//Dozownik 12 (druga faza)                                       			                    
lrDispencer1DoseVolumeShow							:   ST_LrParametr;	 //:=300; 			    // Objętość do wydozowania [ml]
lrDispencer1Phase1VolumeShow						:   ST_LrParametr;	//:=100;			    // Objętość fazy początkowej [ml]
lrDispencer1Phase2VolumeShow						:   ST_LrParametr;	//:=200;			    // Objętość fazy końcowej [ml]
lrDispencer1Phase1VelocityShow						:   ST_LrParametr;	//:=500;			    // Prędkość fazy początkowej [ml/s]
lrDispencer1Phase2VelocityShow						:   ST_LrParametr;	//:=500;			    // Prędkość fazy dozowania [ml/s]
lrDispencer1Phase3VelocityShow						:   ST_LrParametr;	//:=500;			    // Prędkość fazy koncowej [ml/s]
lrDispencer1SuckVelocityShow						:   ST_LrParametr;	//:=500;			    // Prędkość zasysania masy [ml/s2]
lrDispencer1Phase1AccelerationShow					:   ST_LrParametr;	//:=3000;			    // Przyśpieszenie fazy początkowej [ml/s2]
lrDispencer1Phase2AccelerationShow					:   ST_LrParametr;	//:=3000;			    // Przyśpieszenie fazy dozowania [ml/s2]
lrDispencer1Phase3AccelerationShow					:   ST_LrParametr;	//:=3000;			    // Przyśpieszenie fazy końcowej [ml/s2]
lrDispencer1SuckAccelerationShow					:   ST_LrParametr;	//:=3000;			    // Przyśpieszenie zasysania masy [ml/s2]
lrDispencer1Phase1DecelerationShow					:   ST_LrParametr;	//:=3000;			    // Dynamika zwalniania w fazie początkowej
lrDispencer1Phase2DecelerationShow					:   ST_LrParametr;	//:=3000;			    // Dynamika zwalniania dozowania
lrDispencer1Phase3DecelerationShow					:   ST_LrParametr;	//:=3000;			    // Dynamika zwalniania fazy końcowej
udiDispencer1DosingDoneDelayTimeShow				:	ST_UdiParametr; //:=0; 				    // Zwłoka po wydozowaniu
lrDispencer1SuckValveOpenVolumeShow					:   ST_LrParametr;	//:=0;				    // Objętość przy której otwiera się zawór ssania [3] 
lrDispencer1SuckValveOpenTimeDelayShow				:   ST_LrParametr;	//:=0;				    // Zwłoka rozpoczęcia ssania po tłoczeniu [ms] [3]
lrDispencer1SuckValveCloseVolumeShow				:   ST_LrParametr;	//:=0;				    // [H] Objętość zamknięcia zaworu ssania od końca ssania [4]
lrDispencer1SuckValveCloseTimeDelayShow				:   ST_LrParametr;	//:=0;				    // Zwłoka zamknięcia zaworu ssącego [ms] [4] 
lrDispencer1DoseValveOpenVolumeShow					:   ST_LrParametr;	//:=0;				    // [H] Objętość przy której otwiera się zawór tłoczenia [ml] [1]
lrDispencer1DoseValveOpenTimeAccShow				:   ST_LrParametr;	//:=0;				    // Wyprzedzenie otwarcia zaworu tłoczenia [1] [ms]
lrDispencer1DoseValveCloseVolumeShow				:   ST_LrParametr;	//:=0;				    // Pozostała objętość dozy - zamknięcie zaworu tłoczenia [ml] [2]
lrDispencer1DoseValveCloseTimeDecShow				:   ST_LrParametr;	//:=0;				    // Zwłoka zamkniecia zaworu tłoczenia [2] [ms]
lrDispencer1DoseSuckingVolumeShow					:   ST_LrParametr;	//:=0;				    // Ilość dozy do posysenia [ml]	[5] [Podsysanie] 
lrDispencer1DoseSuckingTimeDelayShow				:   ST_LrParametr;	//:=0;				    // Opóźnienie podsysania [ms] [6] [Podsysanie] 
bDispencer1DoseSuckingShow							:	ST_BoolParametr;				        // Aktywacja podsysania
bDispencer1LiftSynchroPh1Show						:	ST_BoolParametr;				        // Synchronizacja z podnosnikiem w fazie początkowej
bDispencer1LiftSynchroPh2Show						:	ST_BoolParametr;				        // Synchronizacja z podnosnikiem w fazie dozowania
bDispencer1LiftSynchroPh3Show						:	ST_BoolParametr;				        // Synchronizacja z podnosnikiem w fazie końcowej
lrDispencer1LifterStartDosePositionShow				:   ST_LrParametr;	//:=20;				    // Pozycja rozpoczęcia dozowania
lrDispencer1LifterStopDosePositionShow				:   ST_LrParametr;	//:=60;				    // Pozycja zakończenia dozowania
lrDispencer1LifterVelocityShow						:   ST_LrParametr;	//:=100;			    // [H] Prędkość podnośnika 
lrDispencer1LifterAccelerationShow					:   ST_LrParametr;	//:=2;				    // [H] Przyspieszenie podnośnika
lrDispencer1LifterDecelerationShow					:   ST_LrParametr;	//:=2;				    // [H] Zwalnianie podnośnika
                                                                                                
//Dozowniki 34 (pierwsza faza)                                                                  		
lrDispencer2DoseVolumeShow							:   ST_LrParametr;	//:=300; 			    // Objętość do wydozowania                                           
lrDispencer2Phase1VolumeShow						:   ST_LrParametr;	//:=100;			    // Objętość fazy początkowej                                         
lrDispencer2Phase2VolumeShow						:   ST_LrParametr;	//:=200;			    // Objętość fazy końcowej                                            
lrDispencer2Phase1VelocityShow						:   ST_LrParametr;	//:=500;			    // Prędkość fazy początkowej                                         
lrDispencer2Phase2VelocityShow						:   ST_LrParametr;	//:=500;			    // Prędkość fazy dozowania                                           
lrDispencer2Phase3VelocityShow						:   ST_LrParametr;	//:=500;			    // Prędkość fazy koncowej                                            
lrDispencer2SuckVelocityShow						:   ST_LrParametr;	//:=500;			    // Prędkość zasysania masy                                           
lrDispencer2Phase1AccelerationShow					:   ST_LrParametr;	//:=3000;			    // Przyspieszenie fazy początkowej                                   
lrDispencer2Phase2AccelerationShow					:   ST_LrParametr;	//:=3000;			    // Przyspieszenie fazy dozowania                                     
lrDispencer2Phase3AccelerationShow					:   ST_LrParametr;	//:=3000;			    // Przyspieszenie fazy końcowej                                      
lrDispencer2SuckAccelerationShow					:   ST_LrParametr;	//:=3000;			    // Przyspieszenie zasysania masy                                     
lrDispencer2Phase1DecelerationShow					:   ST_LrParametr;	//:=3000;			    // Dynamika zwalniania w fazie początkowej                           
lrDispencer2Phase2DecelerationShow					:   ST_LrParametr;	//:=3000;			    // Dynamika zwalniania dozowania                                     
lrDispencer2Phase3DecelerationShow					:   ST_LrParametr;	//:=3000;			    // Dynamika zwalniania fazy końcowej                                 
udiDispencer2DosingDoneDelayTimeShow				:	ST_UdiParametr; //:=0; 				    // Zwłoka po wydozowaniu                                             
lrDispencer2SuckValveOpenVolumeShow					:   ST_LrParametr;	//:=0;				    // Objętość przy której otwiera się zawór ssania [3]                 
lrDispencer2SuckValveOpenTimeDelayShow				:   ST_LrParametr;	//:=0;				    // Zwłoka rozpoczęcia ssania po tłoczeniu [ms] [3]                   
lrDispencer2SuckValveCloseVolumeShow				:   ST_LrParametr;	//:=0;				    // [H] Objętość zamknięcia zaworu ssania od końca ssania [4]    
lrDispencer2SuckValveCloseTimeDelayShow				:   ST_LrParametr;	//:=0;				    // Zwłoka zamknięcia zaworu ssącego [ms] [4]                         
lrDispencer2DoseValveOpenVolumeShow					:   ST_LrParametr;	//:=0;				    // [H] Objętość przy której otwiera się zawór tłoczenia [ml] [1]
lrDispencer2DoseValveOpenTimeAccShow				:   ST_LrParametr;	//:=0;				    // Wyprzedzenie otwarcia zaworu tłoczenia [1] [ms]                   
lrDispencer2DoseValveCloseVolumeShow				:   ST_LrParametr;	//:=0;				    // Pozostała objętość dozy - zamknięcie zaworu tłoczenia [ml] [2]    
lrDispencer2DoseValveCloseTimeDecShow				:   ST_LrParametr;	//:=0;				    // Zwłoka zamkniecia zaworu tłoczenia [2] [ms]                       
lrDispencer2DoseSuckingVolumeShow					:   ST_LrParametr;	//:=0;				    // Ilość dozy do posysenia [ml]	[5] [Podsysanie]                     
lrDispencer2DoseSuckingTimeDelayShow				:   ST_LrParametr;	//:=0;				    // Opóźnienie podsysania [ms] [6] [Podsysanie]                       
bDispencer2DoseSuckingShow							:	ST_BoolParametr;				        // Aktywacja podsysania                                              
bDispencer2LiftSynchroPh1Show						:	ST_BoolParametr;				        // Synchronizacja z podnosnikiem w fazie początkowej                 
bDispencer2LiftSynchroPh2Show						:	ST_BoolParametr;				        // Synchronizacja z podnosnikiem w fazie dozowania                   
bDispencer2LiftSynchroPh3Show						:	ST_BoolParametr;			            // Synchronizacja z podnosnikiem w fazie końcowej                    
lrDispencer2LifterStartDosePositionShow				:   ST_LrParametr;	//:=20;				    // Pozycja rozpoczęcia dozowania                                     
lrDispencer2LifterStopDosePositionShow				:   ST_LrParametr;	//:=60;				    // Pozycja zakończenia dozowania                                     
lrDispencer2LifterVelocityShow						:   ST_LrParametr;	//:=100;			    // [H] Prędkość podnośnika                                      
lrDispencer2LifterAccelerationShow					:   ST_LrParametr;	//:=2;				    // [H] Przyspieszenie podnośnika                                
lrDispencer2LifterDecelerationShow					:   ST_LrParametr;	//:=2;				    // [H] Zwalnianie podnośnika                                    
                                                        		                                
//Chwytak dozowników 1234                                                                       
bDispencersCatchEnableShow	      					:	ST_BoolParametr;			            // [H] Aktywacja    
bDispencersCatchMaxPressureShow	      				:	ST_BoolParametr;			            // Zwiększona siła chwytania            		
lrDispencersCatchHeightSVShow						:   ST_LrParametr;	//:=86;  			    // Pozycja chwytaka
//Kalibracja chwytaków 1234                                                                     
lrDispencersCatch1ClosedValueShow                   :   ST_LrParametr;	                        // Chwytak 1 | wartość kalibracji zamkniętego chwytaka
lrDispencersCatch1OpenValueShow                     :   ST_LrParametr;	                        // Chwytak 1 | wartość kalibracji otwartego chwytaka
lrDispencersCatch2ClosedValueShow                   :   ST_LrParametr;	                        // Chwytak 2 | wartość kalibracji zamkniętego chwytaka
lrDispencersCatch2OpenValueShow                     :   ST_LrParametr;	                        // Chwytak 2 | wartość kalibracji otwartego chwytaka
lrDispencersCatch3ClosedValueShow                	:   ST_LrParametr;	                        // Chwytak 3 | wartość kalibracji zamkniętego chwytaka
lrDispencersCatch3OpenValueShow                     :   ST_LrParametr;	                        // Chwytak 3 | wartość kalibracji otwartego chwytaka
lrDispencersCatch4ClosedValueShow                   :   ST_LrParametr;	                        // Chwytak 4 | wartość kalibracji zamkniętego chwytaka
lrDispencersCatch4OpenValueShow                     :   ST_LrParametr;	                        // Chwytak 4 | wartość kalibracji otwartego chwytaka
lrDispencersCatchToleranceShow                      :   ST_LrParametr;	                        // Tolerancja chwytaka [0-100%]      
                                          		                                                
//Zbiorniki                                                                                     
bTank1MixerEnableShow								:	ST_BoolParametr;	   				    // Mieszadło
bTankHeatingEnableShow								:	ST_BoolParametr;				        // Grzanie                                     		
iTankHeatingTempSVShow								:	ST_DIParametrr;							// Temperatura
bTank1PressureEnableShow							:	ST_BoolParametr;				        // Ciśnienie                                   		
bTank1SupplyPumpEnableShow							:	ST_BoolParametr;			            // Aktywacja pompy 1
bTank2SupplyPumpEnableShow							:	ST_BoolParametr;			            // Aktywacja pompy 2
uTank1LevelSetpointShow								:	ST_UdiParametr;						    // [H] Wartość zadana masy do czujnika poziomu w zbiorniku nr 1
uTank2LevelSetpointShow								:	ST_UdiParametr;						    // [H] Wartość zadana masy do czujnika poziomu w zbiorniku nr 2
bTank1LevelSignalInvertShow							:	ST_BoolParametr;			            // [H] Odwróć sygnał z czujnika zbiornika pierwszego
bTank2LevelSignalInvertShow							:	ST_BoolParametr;			            // [H] Odwróć sygnał z czujnika zbionirka drugiego
                                        			                                            
//Waga                                           			                                    
bWeight1EnableShow									:	ST_BoolParametr;	                    // Aktywacja
lrWeightMassSVShow 									:   ST_LrParametr;						    // Waga zadana 
iWeight1ActuatorUpDelayShow							:	ST_DIParametrr;						    // Opóźnienie podnoszenia wagi 1
iWeight2ActuatorUpDelayShow							:	ST_DIParametrr;						    // Opóźnienie podnoszenia wagi 2
iWeight3ActuatorUpDelayShow							:	ST_DIParametrr;					        // Opóźnienie podnoszenia wagi 3
iWeight4ActuatorUpDelayShow							:	ST_DIParametrr;							// Opóźnienie podnoszenia wagi 4
iWeight5ActuatorUpDelayShow							:	ST_DIParametrr;						    // Opóźnienie podnoszenia wagi 5 
iWeight6ActuatorUpDelayShow							:	ST_DIParametrr;				            // Opóźnienie podnoszenia wagi 6
                                                                                                
//Korekcja wagi                                     			                                
lrFormWeightShow 									:   ST_LrParametr;						    // [H] Waga formatki
lrMass1DensityShow									:   ST_LrParametr;					        // [H] Gęstoć masy pierwszej fazy [g/ml]
lrMass2DensityShow									:   ST_LrParametr;					        // [H] Gęstoć masy drugiej fazy [g/ml]
lrCupWeightShow										:   ST_LrParametr;						    // Waga opakowania (z platynką, zależnie od opakowania) [g]
lrWholePackageWeightShow							:   ST_LrParametr;						    // [H] Waga całego opakowania bez masy (kubeczek,platynka,nakrętka) [g]
lrWeight1MeasurmentCorrectionShow					:   ST_LrParametr;					        // [H] Korekta wagi zmierzonej [g] , różnica pomiedzy wskazaniami wagi zewnętrznej a linią
bDispencer1WeightCorrectionEnableShow				:	ST_BoolParametr;			            // Aktywacja korekcji 1
bDispencer2WeightCorrectionEnableShow				:	ST_BoolParametr;				        // Aktywacja korekcji 2
bDispencer3WeightCorrectionEnableShow				:	ST_BoolParametr;			            // Aktywacja korekcji 3
bDispencer4WeightCorrectionEnableShow				:	ST_BoolParametr;			            // Aktywacja korekcji 4	
lrWeightUpperToleranceShow							:   ST_LrParametr;				            // Górny zakres wagi [g]
lrWeightLowerToleranceShow							:   ST_LrParametr;					        // Dolny zakres wagi [g]
iWeightCorrectionNumberOfSamplesShow				:	ST_UdiParametr;		//:=2;				// Ilość próbek korekcji [x] (1-20)
                                                                                                
//Podajnik platynek                                                                             
bLidFeederEnableShow								:	ST_BoolParametr;			            // Zezwolenie na pracę podajnika platynek 
bLidFeederHeaterEnableShow							:	ST_BoolParametr;		                // Zezwolenie na prace grzałki podajnika platynek 
lrLidFeederHeightPosSVShow							:   ST_LrParametr;						    // Wysokość na której ma znajdować się podajnik platynek
iLidFeederHeatingTimeShow							:	ST_DIParametrr;						    // Czas zgrzewania wstępnego podajnika platynek [ms]
iLidFeederTempHisteresisShow						:	ST_DIParametrr;					        // Histereza poprawnej temperatury grzałki podajnika platynek 1 (+/- *C), po jej przekrocz
iLidFeeder1TempSVShow								:	ST_DIParametrr;						    // Temperatura zadana grzałki podajnika platynek 1
iLidFeeder2TempSVShow								:	ST_DIParametrr;					        // Temperatura zadana grzałki podajnika platynek 2
                                                                                                
//Przeciąganie podajnika platynek                                                               
bLidFeederDragingStationEnableShow					:	ST_BoolParametr;			            // Aktywacja przeciagania formatek pod podajnikem płatynek
lrLidFeederDragingStationVelocityShow				:   ST_LrParametr;	 				        // Prędkosć przeciągania formatek pod podajnikem płatynek [0-100 %]	
lrLidFeederDragingStationAccelerationShow			:   ST_LrParametr;	 				        // Przyspieszenie przeciągania formatek pod podajnikem płatynek 	
lrLidFeederDragingStationDecelerationShow			:   ST_LrParametr;	 				        // Zmniejszenie prędkości przeciągania formatek pod podajnikem płatynek 	
                                                                                                
//Sprawdzanie platynek                                                                          
bLidPuttedCheckEnableShow      						:	ST_BoolParametr;			            	// Zezwolenie na prace stacji sprawdzania nakrętek
lrLidPuttedCheckHeightSVShow 	 					:   ST_LrParametr;	            	        	
lrLidPuttedCheckPositionShow						:   ST_LrParametr;					        	// Pozycka sprawdzania platynki
lrLidPuttedCheckAreaShow							:   ST_LrParametr;					        	// [-50...50]  lrLidPuttedCheckPosition +- lrLidPuttedCheckArea. Granica monitorowania
iLidPuttedCheckProgramShow							:	ST_DIParametrr;								// Program czujnika wizyjnego 0-20
                                                                                                
//Zgrzewanie                                                                                    
bLidSealerEnableShow								:	ST_BoolParametr;			            // Zezwolenie na pracę podajnika 
bLidSealerHeaterEnableShow							:	ST_BoolParametr;			            // Zezwolenie na prace grzałki  
iLidSealerHeatingTimeShow							:	ST_DIParametrr;						    // Czas zgrzewania  [ms]
lrLidSealerPressureShow								:   ST_LrParametr;					        //	Siła zgrzewania [kg] 
lrLidSealerHeightPosSVShow							:   ST_LrParametr;					        // Wysokoć na której ma znajdować się grzałka
iLidSealerTempHisteresisShow						:	ST_DIParametrr;							// Histereza poprawnej temperatury grzałki (+/- *C), po jej przekroczeniu grzałka wpada w 
iLidSealer1TempSVShow								:	ST_DIParametrr;					        // Temperatura zadana grzałki 1                                                           
iLidSealer2TempSVShow								:	ST_DIParametrr;				            // Temperatura zadana grzałki 2
                                                                                                
//Przeciąganie zgrzewania                                                                       
bLidSealerDragingStationEnableShow					:	ST_BoolParametr;			            // Aktywacja przeciagania formatek pod zakrecarkami
lrLidSealerDragingStationVelocityShow				:   ST_LrParametr;				            // Prędkosć przeciągania formatek pod zakręcarkami [0-100 %]
lrLidSealerDragingStationAccelerationShow			:   ST_LrParametr;	 				        // Przyspieszenie przeciągania formatek pod podajnikem płatynek 	
lrLidSealerDragingStationDecelerationShow			:   ST_LrParametr;					        // Zmniejszenie prędkości przeciągania formatek pod podajnikem płatynek 	
                                                                                                
//Szlaban podawania zamknięć                            				                        
bCapFeederGateEnableShow							:	ST_BoolParametr;		                // Aktywacja 
iCapFeederGateBlockingTimeShow						:	ST_DIParametrr;							// Czas blokowania
                                                                                                
//[H] Podajnik zamknięć                        				                                    
bCapFeederEnableShow								:	ST_BoolParametr;		                // [H] Aktywacja
lrCapFeederHeightPosSVShow							:   ST_LrParametr;	//:=140;			    // [H] Pozycja
iCapFeederTimeDelayOnShow							:	ST_DIParametrr;						    // [H] Opóźnienie włączenia
iCapFeederTimeDelayOffShow							:	ST_DIParametrr;						    // [H] Opóźnienie wyłączenia
iCapFeederTimeToEmptySleeveErrorShow				:	ST_DIParametrr;						    // [H] Czas do alarmu pustego rękawa [s] (10-120 s)
                                                                                                
//Sorter nasadek                                                                                
//Zmienne z innego sterownika                                                                   
bCapSorterOnlyWeightOKEnableShow					:	ST_BoolParametr;		                // Nakładanie zamknięć tylko na opakowania z waga OK
                                                                                                
//Przeciąganie pod sorterem nasadek                                                             
bCapSorterDragEnableShow							:	ST_BoolParametr;		                // [H] Aktywacja
lrCapSorterDragVelocityShow							:   ST_LrParametr;					        // Prędkość
lrCapSorterDragAccelerationShow						:   ST_LrParametr;						    // Przyspieszenie 
lrCapSorterDragDecelerationShow						:   ST_LrParametr;					        // Hamowanie
                             				                                                    
//Sprawdzanie nasadki                                      				                        
bCapPuttedCheckEnableShow							:	ST_BoolParametr;			            // Aktywacja
lrCapPuttedCheckHeightPosSVShow						:   ST_LrParametr;	//:=69;				    // Pozycja
                             					                                                
//Zakrecarka szczekowa (Zachować kolejność i opisy!)                                            
bGripperScrewer1EnableShow							:	ST_BoolParametr;			            // Aktywacja 1
lrGripperScrewingTightTorqueShow					:   ST_LrParametr;	  				        // Nastawa momentu zakręcania [Nm]
bGripperScrewer2EnableShow							:	ST_BoolParametr;		                // Aktywacja 2
lrGripperScrewing2TightTorqueShow					:   ST_LrParametr;	  				        // Nastawa momentu zakręcania 2 [Nm]
iGripperScrewer1ToolShow							:	ST_DIParametrr;					        // Wybór narzędzia (1-5), opisy w tablicy AsGripperScrewerTool	
lrGripperScrewer1VelocityShow						:   ST_LrParametr;	//:=6000; 			    // Prędkość zakręcania [rpm]
nGripperScrewer1TightTimeShow						:	ST_DiParametrr; //:=100;  			    // Czas przytrzymania podczas dokręcania [ms] 	
iGripperScrewer1StartDelayShow						:	ST_DIParametrr;					        // Zwoka przed zakręcaniem			
lrGripperScrewerReadyPositionShow					:   ST_LrParametr;	 //:= 250;  		    // Pozycja gotowości
lrGripperScrewerPushingCapPositionShow				:   ST_LrParametr;	//:= 250;  		        // Pozycja docisku  
lrGripperScrewerScrewingCapPositionShow				:   ST_LrParametr;	//:= 250;  		        // Pozycja zakręcania	
lrGripperScrewerPressureShow						:   ST_LrParametr;						    // Siła chwytaka nasadki (0.0 kg)
lrGripperScrewerCatchPressureShow 					:   ST_LrParametr;						    // Siła chwytaka butelki (0.0 kg)
lrDispencerCatchPressureShow 						:   ST_LrParametr;						    // Siła chwytaka butelki pod dozownikami (0.0 kg)
lrGripperScrewerPressureExhaustLevelShow			:   ST_LrParametr;						    // Prędkość zamykania chwytaka nasadki (0.0-100.0 %)
lrGripperScrewerCatchPressureExhaustLevelShow		:   ST_LrParametr;						    // Prędkość zamykania chwytaka opakowania (0.0-100.0 %)
lrGripperScrewerTurnoversToFullScrewedShow			:   ST_LrParametr;						    // Opakowanie | Ilość obrotów zamknięcia [obr.] (0.5-10.0 obr.)
lrGripperScrewerThreadPitchShow						:   ST_LrParametr;						    // Opakowanie | Skok gwintu [mm] (0.1-10.0 mm)
lrGripperScrewerThreadTimesShow						:   ST_LrParametr;						    // Opakowanie | Krotność gwintu [x] (1-10 x)                       		
nGripperScrewerCatchHeightSVShow					:	ST_DiParametrr; //:=86;  				// Pozycja chwytaka opakowań
bGripperScrewer1FindScrewShow						:	ST_BoolParametr;			            // Szukanie gwintu w pozycji zakręcania	
bGripperScrewer1Option4Show							:	ST_BoolParametr;			            // Szukanie gwintu w pozycji dociskania	
lrGripperScrewer1FindingScrewDegreeShow				:   ST_LrParametr;	 				        // Kąt szukania gwintu (max. dla opcji szukania gwintu z czuj. wys.)	
bGripperScrewer1Option1Show							:	ST_BoolParametr;		                // Otwarty chwytak przy szukaniu gwintu	
bGripperScrewer1Option2Show							:	ST_BoolParametr;			            // Obrót do tyłu w pozycji dociskania (w trakcie przejazdu do poz. doc.)
bGripperScrewer1Option3Show							:	ST_BoolParametr;			            // Dodatkowy ruch chwytakiem przed zakręceniem  (w poz. doc.)	
bGripperScrewer1Option5Show							:	ST_BoolParametr;			            // Szukanie gwintu z czujnikiem wysokości
bGripperScrewer1Option6Show							:	ST_BoolParametr;			            // Obrót z pozycji docisku do zakręcania
bGripperScrewer1Option7Show							:	ST_BoolParametr;		                // Tryb momentowy	
                                                                                                
//Przeciaganie formatek pod zakrecarkami                                                        
bBottleDragingStationEnableShow						:	ST_BoolParametr;			            // [H] Aktywacja 
lrBottleDragingStationVelocityShow					:   ST_LrParametr;					        // Prędkość
                                                                                                
//Sprawdzanie zakręcania                                                                        
bCapCorrectCheckEnableShow							:	ST_BoolParametr;				        // Aktywacja
lrCapCorrectCheckHeightPosSVShow					:   ST_LrParametr;	//:=69;				    // Pozycja
bCapCorrectCheckCameraEnableShow      				:	ST_BoolParametr;			            // Aktywacja sprawdzania orientacji nasadki
iCapCorrectCheckCameraProgramShow					:	ST_DIParametrr;			                // Program czujnika wizyjnego 0-20
                                                                                                
                                                                                                
//Robot butelek                                                                                 
bBottleTransferEnableShow							:	ST_BoolParametr;			            // Aktywacja
nBottleTransferProgramShow							:	ST_UdiParametr;						    // [H] Program robota	
iBottleTransferPickOffsetXShow 						:	ST_DIParametrr;					        // Offset X pozycji pobrania
iBottleTransferPickOffsetYShow 						:	ST_DIParametrr;							// Offset Y pozycji pobrania  
iBottleTransferPickOffsetZShow 						:	ST_DIParametrr;							// Offset Z pozycji pobrania
iBottleTransferPick2OffsetXShow						:	ST_DIParametrr;							// Offset X 2 pozycji pobrania	
iBottleTransferPick2OffsetYShow						:	ST_DIParametrr;					        // Offset Y 2 pozycji pobrania
iBottleTransferPick2OffsetZShow						:	ST_DIParametrr;							// Offset Z 2 pozycji pobrania
iBottleTransferPlace1OffsetXShow 					:	ST_DIParametrr;							// Offset X pozycji etykieciarki
iBottleTransferPlace1OffsetYShow 					:	ST_DIParametrr;							// Offset Y pozycji etykieciarki
iBottleTransferPlace1OffsetZShow 					:	ST_DIParametrr;						    // Offset Z pozycji etykieciarki
iBottleTransferPlace2OffsetXShow 					:	ST_DIParametrr;							// Offset X pozycji odrzutu
iBottleTransferPlace2OffsetYShow					:	ST_DIParametrr;							// Offset Y pozycji odrzutu	
iBottleTransferPlace2OffsetZShow 					:	ST_DIParametrr;							// Offset Z pozycji odrzutu
iBottleTransferSpeedShow							:	ST_DIParametrr;	  //:= 10;			    // Prędkość robota 	
bBottleTransferInkJetEnableShow						:	ST_BoolParametr;			            // Przesuwanie opakowania nad drukarką (Inkjet)
bBottleTransferPickOnlyOneShow						:	ST_BoolParametr;			            // [H] Pobieranie tylko 1 opakowania
bBottleTransferWeightEnableShow						:	ST_BoolParametr;				        // Przesuwanie opakowania na wagę 
iBottleTransferWeightIntervalShow					:	ST_DIParametrr;							// Interwał przesuwania na wagę
bBottleTransferRotateEnableShow						:	ST_BoolParametr;                        // Obrót orientacji nasadki   
                                                                                                
//Transporter odrzutu                      	                                                    
bBadBottleConveyorEnableShow						:	ST_BoolParametr;				        // [H] Aktywacja
nBadBottleConveyorVelocitySVShow					:	ST_UdiParametr;						    // Prędkość
                                                                                                
//Etykieciarka                                                                                  
bLabelMachineEnableShow								:	ST_BoolParametr;				        // Aktywacja
                                                                                                
//Stół odbierający                                                                              
bExitTurnTable1EnableShow							:	ST_BoolParametr;				        // Aktywacja
//Transporter odbierający                                                                       
bExitConveyorEnableShow								:	ST_BoolParametr;			            // Aktywacja
nExitConveyorVelocitySVShow							:	ST_UdiParametr;						    // Prędkość
                                                                                                
                                                                                                
//Transportery główne                                                                           
bFormTransportersEnableShow							:	ST_BoolParametr;				        // [H] Aktywacja
nFormTransportersDispencerVelocitySVShow			:	ST_UdiParametr;				            // Prędkość transportera przed dozownikami
nFormTransportersScrewerVelocitySVShow				:	ST_UdiParametr;				            // Prędkość transportera za dozownikami
nFormTransportersBeforeScrewerVelocitySVShow		:	ST_UdiParametr;			                // Prędkość transportera przed zakręcarką
nFormTransportersSlowerVelocitySVShow				:	ST_UdiParametr;				            // Prędkość spowalniacza 
                                                                                                
                                                                                                
//[H] InkJet obwodowy                                                                           
bCircularInkjetEnableShow							:	ST_BoolParametr;				        // [H] Aktywacja
iCircularInkjetSpeedShow							:	ST_DIParametrr;							// [H] Prędkość 
iCircularInkjetDelayShow							:	ST_DIParametrr;							// [H] Opóźnienie docisku rolek
iCircularInkjetHoldShow								:	ST_DIParametrr;							// [H] Czas przytrzymania [ms]

bROPPCappingEnableShow 								:	ST_BoolParametr;	
bROPPDragEnableShow 								:	ST_BoolParametr;	
bROPPFeederEnableShow 								:	ST_BoolParametr;	
bROPPSlowerEnableShow 								:	ST_BoolParametr;	
iROPPCapping1ToolShow 								:	ST_DIParametrr;	
iROPPCappingTime2Show 								:	ST_DIParametrr;	
iROPPCappingTimeShow 								:	ST_DIParametrr;	
iROPPFeederTimeDelayOffShow							:	ST_DIParametrr;	
iROPPFeederTimeDelayOnShow 							:	ST_DIParametrr;	
iROPPFeederTimeToEmptySleeveErrorShow 				:	ST_DIParametrr;	
lrROPPCappingHeightPosSVShow						:	ST_LrParametr;	
lrROPPCappingVelocitySVShow 						:	ST_LrParametr;	
lrROPPDragAccelerationShow 							:	ST_LrParametr;	
lrROPPDragDecelerationShow 							:	ST_LrParametr;	
lrROPPDragVelocityShow 								:	ST_LrParametr;	
lrROPPFeederHeightPosSVShow 						:	ST_LrParametr;	                                                                             
nROPPSlowerVelocitySVShow 							:	ST_UdiParametr;	

END_STRUCT                                                                                      
END_TYPE

// ---- POUs/Recipes/NewRecipes/ST_Recipe_UCF_PARAM.TcDUT
TYPE ST_Recipe_UCF_PARAM :
STRUCT
		//Sorter nasadek, typ produktu	
	iCapSorterProductType										:	ST_DIParametrr;		//:= 2; 		//		Typ produktu: 0- kule/fliptopy, 1- pompki, 2- disctop, 3-airless, 4-decoration cap (wyłączone podcisnienie na załapywarce), 5- decoration cap with new gripper (wyłączone podcisnienie + nowy program do robota)
	uiCapSorterIndexShow										:	ST_UdiParametr;	//:= 5;		//		Index produktu	
	bPresenceBottleEnableShow									:	ST_BoolParametr;					//		Sprawdzanie butelki w formatce

//--------------------------------------CapSorterTransporter-----------------------------------------------------------------------------------------------------------------------------	
	// Sorter nasadek, transporter zasobnika
	bCapSorterTransporterEnableShow								:	ST_BoolParametr;				//		Aktywacja
	iCapSorterTransporterTankConveyorVelocityShow				:	ST_DIParametrr;		//:= 1200;	//		Prędkość 							| [%] (1.0-100.0)
	iCapSorterTransporterStartDelayTimeShow						:	ST_DIParametrr;		//:= 100;		//		Timer do załączania 				| [ms] (0.0-10_000.0)
	udiCapSorterTransporterTimeProductOnSensorBeforeBrushShow	:	ST_UdiParametr;		//:= 150;		//		Timer pracy							| [ms] (0.0-10_000.0)
	iCapSorterTransporterEmptyingConveyorSpeedShow				:	ST_DIParametrr;		//:= 25;		// 		Prędkość, opróżnianie 				| [%] (1.0-100.0)
	iCapSorterTransporterVolumeOfCapsShow						:	ST_DIParametrr;		//:= 330;		//		Odłegłość do zamknięć, ostrzeżenie 	| [mm] (0.0-10_000.0)

//---------------------------------------CapSorterWheel----------------------------------------------------------------------------------------------------------------------------	
	// Sorter nasadek, stól
	bCapSorterWheelEnableShow									:	ST_BoolParametr;				//		Aktywacja
	lrCapSorterWheelMoveAccelerationEmptyTableShow				:   ST_LrParametr;			//:= 5000;	//		Dynamika rozpędzania - pusty 		| [obr/min²], (1.0-100_000.0) 
	lrCapSorterWheelMoveDecelerationEmptyTableShow				:   ST_LrParametr;			//:= 5000;    //		Dynamika spowalniania - pusty 		| [obr/min²] (1.0-100_000.0) 
	lrCapSorterWheelMoveSpeedEmptyTableShow						:   ST_LrParametr;		//:= 334;     //		Prędkość - pusty 					| [obr/min] (1.0-10_000.0)                
	lrCapSorterWheelMoveAngleEmptyTableShow						:   ST_LrParametr;			//:= 20;      //		Kąt - pusty 						| [obr/min] (0.0-360.0)                        
	lrCapSorterWheelJerkAngleEmptyTableShow						:   ST_LrParametr;		//:= 15000;   //		Zryw - pusty 						| [obr/min³] (1.0-1_000_000)                  
	iCapSorterWheelWaitingAfterRotationEmptyTableShow			:	ST_DIParametrr;		//:= 100;     //		Czas stabilizacji - pusty 			| [ms] (0.0-1_000)                 
	                                                                        //
	lrCapSorterWheelMoveAccelerationFullTableShow				:   ST_LrParametr;		//:= 5000;	//		Dynamika rozpędzania - pełny 		| [obr/min²], (1.0-100_000.0) 
	lrCapSorterWheelMoveDecelerationFullTableShow				:   ST_LrParametr;		//:= 5000;    //		Dynamika spowalniania - pełny 		| [obr/min²] (1.0-100_000.0) 
	lrCapSorterWheelMoveSpeedFullTableShow						:   ST_LrParametr;		//:= 334;     //		Prędkość - pełny 					| [obr/min] (1.0-10_000.0)                
	lrCapSorterWheelMoveAngleFullyTableShow						:   ST_LrParametr;			//:= 6;       //		Kąt - pełny 						| [obr/min] (0.0-360.0)                        
	lrCapSorterWheelJerkAngleFullTableShow						:   ST_LrParametr;			//:= 15000;   //		Zryw - pełny 						| [obr/min³] (1.0-1_000_000)                  
	iCapSorterWheelWaitingAfterRotationFullTableShow			:	ST_DIParametrr;		//:= 30;      //		Czas stabilizacji - pełny 			| [ms] (0.0-1_000)                 
	                                                                        //
	lrCapSorterWheelMoveAccelerationHalfFullTableShow			:   ST_LrParametr;			//:= 5000;	//		Dynamika rozpędzania - półpełny 	| [obr/min²], (1.0-100_000.0) 
	lrCapSorterWheelMoveDecelerationHalfFullTableShow			:   ST_LrParametr;			//:= 5000;    //		Dynamika spowalniania - półpełny 	| [obr/min²] (1.0-100_000.0) 
	lrCapSorterWheelMoveSpeedHalfFullTableShow					:   ST_LrParametr;			//:= 334;     //		Prędkość - półpełny 				| [obr/min] (1.0-10_000.0)                
	lrCapSorterWheelMoveAngleHalfFullyTableShow					:   ST_LrParametr;			//:= 12;      //		Kąt - półpełny						| [obr/min] (0.0-360.0)                        
	lrCapSorterWheelJerkAngleHalfFullTableShow					:   ST_LrParametr;			//:= 15000;   //		Zryw - półpełny 					| [obr/min³] (1.0-1_000_000)                  
	iCapSorterWheelWaitingAfterRotationHalfFullTableShow		:	ST_DIParametrr;		//:= 50;      //		Czas stabilizacji - półpełny 		| [ms] (0.0-1_000)                 

//-------------------------------------CapSorterCamera------------------------------------------------------------------------------------------------------------------------------	                                                    	
	// Sorter nasadek, system wizyjny
	
    bCapSorterCameraEnableShow									:	ST_BoolParametr;				//	[H]	Aktywacja                            	
	
//-----------------------------------------CapSorterRobot--------------------------------------------------------------------------------------------------------------------------	
	// Sorter nasadek, robot
	bCapSorterRobotEnableShow									:	ST_BoolParametr;				//		Aktywacja
                                                                                                                           	
	lrCapSorterRobotPlace1PositionXShow							:   ST_LrParametr;					//		Offset odkładania 1, X 			| [mm]	((-100.0)-100.0)       
	lrCapSorterRobotPlace1PositionYShow							:   ST_LrParametr;	    			//		Offset odkładania 1, Y 			| [mm]	((-100.0)-100.0)       
	lrCapSorterRobotPlace1PositionZShow							:   ST_LrParametr;	    			//		Offset odkładania 1, Z 			| [mm]	((-100.0)-100.0)       
	lrCapSorterRobotPlace1PositionCShow							:   ST_LrParametr;	    			//		Offset odkładania 1, C 			| [° ]	((-360.0)-360.0)                 
	iCapSorterRobotPickElevationShow							:	ST_DIParametrr;				//		Punkt nad poz. Pick				| [mm]	(30-1000)
	iCapSorterRobotPickTimeShow									:	ST_DIParametrr;					//		Czas przyssania					| [ms]	(0-10_000)
	iCapSorterRobotVacuumActivationShow							:	ST_DIParametrr;					//		Czas przed przyssaniem			| [ms]	(0-1000)
	iCapSorterRobotVacuumOffShow								:	ST_DIParametrr;					//		Czas przed oddmuchem			| [ms]	(0-1000)
	iCapSorterRobotPlaceTimeShow								:	ST_DIParametrr;					//		Czas oddmuchu					| [ms]	(0-1000)
	iCapSorterRobotTCP_PlaceOffsetShow							:	ST_DIParametrr;					//		Wysokość od TCP do p. odłożenia	| [mm]	(0-1000)									
	iCapSorterRobotAccelerationDecelerationShow					:	ST_DIParametrr;					//		Dynamika rozpędzania/hamowania	| [%]	(20-100)
	iCapSorterRobotGripperWatchdogShow							:	ST_DIParametrr;					//		Czas sprawdzania silownika		| [ms]	(0-1000)
	iCapSorterRobotParalaxCorrectionShow						:	ST_DIParametrr;				//		Korekta paralaxy				| [mm]	(0-100)
	
	iCapSorterRobotNumberToolShow								:	ST_DIParametrr;				//		Numer narzędzia					| 		(0-10)
	iCapSorterRobotPickPositionZShow							:	ST_DIParametrr;					//		Wysokość pobierania 			| [mm]	(0-200)
	iCapSorterRobotTCP_Lenght									:	ST_DIParametrr;					//		Długość chwytaka				| [mm]	(10-100)
	iCapSorterRobotProductDiametr								:	ST_DIParametrr;					//		Średnica nasadki				| [mm] 	(10-100)
	
//----------------------------------------CapSorterIntermediateTransporter---------------------------------------------------------------------------------------------------------------------------
	// Sorter nasadek, transporter zasypowy
	bCapSorterIntermediateTransporterEnableShow					:	ST_BoolParametr;			//		Aktywacja
	iCapSorterIntermediateTransporterAutoSpeedShow				:	ST_DIParametrr;		//:= 20;		//		Prędkość 					| [%] (1.0-100.0)
	iCapSorterIntermediateTransporterManualSpeedShow			:	ST_DIParametrr;		//:= 30;		//		Prędkość, manual 			| [%] (1.0-100.0)
	iCapSorterIntermediateTransporterEmptyingSpeedShow			:	ST_DIParametrr;		//:= 50;		//		Prędkość, opróżnianie 		| [%] (1.0-100.0)
	iCapSorterIntermediateTransporterDelayCountTimeShow			:	ST_DIParametrr;		//:= 100;		//		Timer pracy					| [ms]	(0.0-100_000.0)
	iCapSorterIntermediateTransporterReverseTimeShow			:	ST_DIParametrr;		//:= 4000;	//		Timer odwróconej pracy 		| [ms] (0.0-10_000.0)
	udiCapSorterIntermediateTransporterTimeProductOnSensorShow	:	ST_UdiParametr;		//:= 1800;	//		Czas produktu na czujniku 	| [ms] (0.0-10_000.0)	
	lrCapSorterIntermediateTransporterWheelAngleShow			:   ST_LrParametr;			//:= 6;		//		Kąt zasypu 					| [°] (1.0-360.0)
	
//----------------------------------------CapSorterIntermediateBrush---------------------------------------------------------------------------------------------------------------------------
	//Sorter nasadek, szczotka transportera
	bCapSorterIntermediateBrushEnableShow						:	ST_BoolParametr;				//		Aktywacja
	iCapSorterIntermediateBrushAutoSpeedShow					:	ST_DIParametrr;		//:= 30;		//		Prędkość  					| [%] (0.0-100.0)
	iCapSorterIntermediateBrushManualSpeedShow					:	ST_DIParametrr;		//:= 30;		//		Prędkość, manual 			| [%] (0.0-100.0)
	iCapSorterIntermediateBrushEmptyingSpeedShow				:	ST_DIParametrr;		//:= 30;		//		Prędkość, opróżnianie 		| [%] (0.0-100.0)
	lrCapSorterIntermediateBrushPositionHeightSVShow			:   ST_LrParametr;			//:= 45;		//		Wysokość 					| [mm] (0.0-10_000.0)

//----------------------------------------CapSorterBrush1OnWheel---------------------------------------------------------------------------------------------------------------------------
	// Sorter nasadek, szczotka stolu 1
	bCapSorterBrush1OnWheelEnableShow							:	ST_BoolParametr;					//		Aktywacja
	iCapSorterBrush1OnWheelAutoSpeedShow						:	ST_DIParametrr;		//:= 30;		//		Prędkość 					| [%] (0.0-100.0)
	iCapSorterBrush1OnWheelManualSpeedShow						:	ST_DIParametrr;		//:= 30;		//		Prędkość, manual 			| [%] (0.0-100.0)
	iCapSorterBrush1OnWheelEmptyingSpeedShow					:	ST_DIParametrr;		//:= 30;		//		Prędkość, opróżnianie 		| [%] (0.0-100.0)
	lrCapSorterBrush1OnWheelPositionHeightSVShow				:   ST_LrParametr;			//:= 45;		//		Wysokość 					| [mm] (0.0-10_000.0)
	
//----------------------------------------CapSorterBrush2OnWheel----------------------------------------------------------------------------------
	// Sorter nasadek, szczotka stolu 2
	bCapSorterBrush2OnWheelEnableShow							:	ST_BoolParametr;					//		Aktywacja
	iCapSorterBrush2OnWheelAutoSpeedShow						:	ST_DIParametrr;		//:= 30;		//		Prędkość 					| [%] (0.0-100.0)
	iCapSorterBrush2OnWheelManualSpeedShow						:	ST_DIParametrr;		//:= 30;		//		Prędkość, manual 			| [%] (0.0-100.0)
	iCapSorterBrush2OnWheelEmptyingSpeedShow					:	ST_DIParametrr;		//:= 30;		//		Prędkość, opróżnianie 		| [%] (0.0-100.0)
	lrCapSorterBrush2OnWheelPositionHeightSVShow				:   ST_LrParametr;		//:= 45;		//		Wysokość 					| [mm] (0.0-10_000.0)

//------------------------------------------CapFeeder-------------------------------------------------------------------------------------------------------------------------	
	// Sorter nasadek, 
	bCapSorterFeederEnableShow									:	ST_BoolParametr;				//		Aktywacjaa
	bCapSorterFeederEnableTubeError								:	ST_BoolParametr;				// 		Aktywacja błedu słomki
	lrCapSorterFeederMover1InputPositionShow					:   ST_LrParametr;					//		Pozycja wkładania, wózek 1 	| [mm] (?-?)
	lrCapSorterFeederMover2InputPositionShow					:   ST_LrParametr;					//		Pozycja wkładania, wózek 2 	| [mm] (?-?)
	lrCapSorterFeederMover1OutputPositionShow					:   ST_LrParametr;					//		Pozycja wyjmowania, wózek 1 | [mm] (?-?)
	lrCapSorterFeederMover2OutputPositionShow					:   ST_LrParametr;					//		Pozycja wyjmowania, wózek 2 | [mm] (?-?)
	lrCapSorterFeederSlotDistanceShow							:   ST_LrParametr;					//		Offset wkładania			| [mm] (?-?)			Old-(Odstęp między pozycjami kładzenia)
	lrCapSorterFeederMoverSpeedShow								:   ST_LrParametr;					//		Prędkość				 	| [%] (0.0-100.0)
	lrCapSorterFeederMoverAccelerationShow						:   ST_LrParametr;					//		Przyspieszenie 				| [mm/s²] 
	lrCapSorterFeederMoveJerkShow								:   ST_LrParametr;				//		Zryw						| [mm/s³]

//-------------------------------------------------------------------------------------------------------------------------------------------------------------------	
	//CapPreScrewer		
	bCapSorterPreScrewerEnableShow								:	ST_BoolParametr;				// 		Aktywacja
	bCapSorterPreScrewerPicker1EnableShow						:	ST_BoolParametr;			// 		Aktywacja	
	bCapSorterPreScrewerPicker2EnableShow						:	ST_BoolParametr;			// 		Aktywacja
	bCapSorterPreScrewerPicker3EnableShow						:	ST_BoolParametr;				// 		Aktywacja	
	bCapSorterPreScrewerPicker4EnableShow						:	ST_BoolParametr;				// 		Aktywacja
	//Oś Z
	lrCapSorterPreScrewerPickZPositionShow						:   ST_LrParametr;					//		Wysokość pobierania						| [mm]	
	lrCapSorterPreScrewerCatcherReleseShow						:   ST_LrParametr;					//		nie używamy Wysokość otwierania chwytaka nakrętek	| [mm]		
	lrCapSorterPreScrewerCapCatcherZPositionShow				:   ST_LrParametr;					//		Wysokość zamykania nakrętkek			| [mm]
	lrCapSorterPreScrewerTopZPositionShow						:   ST_LrParametr;					//		Pozycja górna ośi Z						| [mm] 	
	lrCapSorterPreScrewerCartesianCatchZPositionShow			:   ST_LrParametr;	 				//      Wait Position
	lrCapSorterPreScrewerStrawCatcherZPositionShow				:   ST_LrParametr;					//		Wysokość otwierania łapaczy słomek		| [mm]	
	LrCapSorterPreScrewerCheckStrawCatcherActuatorZPosition		:   ST_LrParametr;					//		Wysokość sparawdzania cofania łapaczy słomek	| [mm]	
	lrCapSorterPreScrewerScrewerStartZPositionShow				:   ST_LrParametr;					//		Wysokość początku zakręcania			| [mm]	
	lrCapSorterPreScrewerGripperOpenPositionShow				:   ST_LrParametr;					//		Pozycja otwierania chwytaka butelek 	| [mm]
	lrCapSorterPreScrewerPlaceZPositionShow						:   ST_LrParametr;					//		Wysokość odkładania - koniec załapywania gwintu	| [mm]   	
	//Wspólne ruchi	
	lrCapSorterPreScrewerBendingDistanceShow					:   ST_LrParametr;					//		Odległość zaokrąglania ruchów 			| [mm]		
	lrCapSorterPreScrewerStrawInsertDistance					:   ST_LrParametr;					//		Odległość wspólnego ruchu, prowadzenie słomki	| [mm]		
	//Oś x
	lrCapSorterPreScrewerPickXMover1PositionShow				:   ST_LrParametr;				//		Pozycja osi poziomej do pobierania, wozek 1	| [mm]
	lrCapSorterPreScrewerPickXMover2PositionShow				:   ST_LrParametr;					//		Pozycja osi poziomej do pobierania, wozek 2	| [mm]
	lrCapSorterPreScrewerPlaceXPositionShow						:   ST_LrParametr;			//		Pozycja osi poziomej do odkładania			| [mm]
	//Oś zakręcania
	lrCapSorterPreScrewerScrewFindingShow						:   ST_LrParametr;					//		Kąt szukania gwintu							| [°]
	lrCapSorterPreScrewerScrewDistanceShow						:   ST_LrParametr;					//		Kąt zakręcania								| [°]
	//Prédkośći                                                                                                                         	
	lrCapSorterPreScrewerPickerSpeedShow						:   ST_LrParametr;					//		Prędkość									| [mm/s]   
	lrCapSorterPreScrewerPickerAccelerationShow					:   ST_LrParametr;				//		Przyspieszenie								| [mm/s²] 		
	lrCapSorterPreScrewerPickerJerkShow							:   ST_LrParametr;					//		Zryw										| [mm/s³]
                                                                                                                                        	
	lrCapSorterPreScrewerCatcherSpeedShow						:   ST_LrParametr;					//		Prędkość									| [mm/s] 
	lrCapSorterPreScrewerCatcherAccelerationShow				:   ST_LrParametr;					//		Przyspieszenie								| [mm/s²] 	
	lrCapSorterPreScrewerCatcherJerkShow						:   ST_LrParametr;					//		Zryw										| [mm/s³]	                                                                                                                                 	
	lrCapSorterPreScrewerScrewSpeedShow							:   ST_LrParametr;					//		Prędkość zakręcania							| [mm/s]
	lrCapSorterPreScrewerScrewAccelerationShow					:   ST_LrParametr;					//		Przyspieszenie zakręcania				| [mm/s²]
	lrCapSorterPreScrewerScrewJerkShow							:   ST_LrParametr;				//		Zryw zakręcania							| [mm/s³]

	//Oś łapacza słomki	
	lrCapSorterPreScrewerCatcherCatchingPositionShow			:   ST_LrParametr;					//		Pozycja łapania słomki					| [mm]
	lrCapSorterPreScrewerCatcherPlacePositionShow				:   ST_LrParametr;					//		Pozycja dolna łapacza słomki			| [mm]
	lrCapSorterPreScrewerCatcherHightSVShow						:   ST_LrParametr;					//		Nastawa wysokości stacji łapacza słomek		| [mm]
	//Kalibracja chwytaków butelki
	bCapSorterPreScrewerBottleCatcherEnableShow					:	ST_BoolParametr;			//		Actywacja chwytaków butelki
	lrCapSorterPreScrewerBottleCatch1OpenValueShow				:   ST_LrParametr;					//		Chwytak 1 | wartość kalibracji otwartego chwytaka
	lrCapSorterPreScrewerBottleCatch1CloseValueShow				:   ST_LrParametr;					//		Chwytak 1 | wartośc kalibracji zamkniętego chwytaka
	lrCapSorterPreScrewerBottleCatch2OpenValueShow				:   ST_LrParametr;					//		Chwytak 2 | wartość kalibracji otwartego chwytaka
	lrCapSorterPreScrewerBottleCatch2CloseValueShow				:   ST_LrParametr;					//		Chwytak 2 | wartość kalibracji zamkniętego chwytaka
	lrCapSorterPreScrewerBottleCatch3OpenValueShow				:   ST_LrParametr;	                //		Chwytak 3 | wartość kalibracji otwartego chwytaka
	lrCapSorterPreScrewerBottleCatch3CloseValueShow				:   ST_LrParametr;					//		Chwytak 3 | wartość kalibracji zamkniętego chwytaka	
	lrCapSorterPreScrewerBottleCatch4OpenValueShow				:   ST_LrParametr;	                //		Chwytak 4 | wartość kalibracji otwartego chwytaka
	lrCapSorterPreScrewerBottleCatch4CloseValueShow				:   ST_LrParametr;					//		Chwytak 4 | wartość kalibracji zamkniętego chwytaka
	                                                        	
	lrCapSorterPreScrewerBottleCatchToleranceValueShow			:   ST_LrParametr;				//		Tolerancja chwytaków
	lrCapSorterPreScrewerCatchAngleOpenSV						:   ST_LrParametr;		//:= 180.0;		//		[] Kąt puszczania centrowników
	
	lrCapSorterPreScrewerWaitInPlaceTimeShow					:   ST_LrParametr;		//:= 50;			//		Czas zatrzymania w miejscu odłożenia 	| [ms]
	
	bCapSorterPreScrewerCatchAngleOpenEnaShow					:	ST_BoolParametr;					// 		Aktywacja puszczania centrowników po osiągnięciu zadanego kątu
	bCapSorterPreScrewerPoundedInCap							:	ST_BoolParametr;				// 		Wbijana nasadka
	
//Parametry do obliczeń 
	lrCapSorterBottleHightShow									:   ST_LrParametr;					//		Wysokość butelki
	lrCapSorterBottleNeckHightShow								:   ST_LrParametr;					// 		Wysokość szyjki butelki
	lrCapSorterCapHightShow										:   ST_LrParametr;					// 		Wysokość zamknięcia
	lrCapSorterCapNeckHightShow									:   ST_LrParametr;					//		Wysokość szyjki zamknięcia

//Rezerwa	
	lrCapSorterSpare1											:   ST_LrParametr;					//Rezerwa 1
	lrCapSorterSpare2											:   ST_LrParametr;					//Rezerwa 2
	lrCapSorterSpare3											:   ST_LrParametr;					//Rezerwa 3
	lrCapSorterSpare4											:   ST_LrParametr;					//Rezerwa 4
	lrCapSorterSpare5											:   ST_LrParametr;					//Rezerwa 5
	lrCapSorterSpare6											:   ST_LrParametr;					//Rezerwa 6
	lrCapSorterSpare7											:   ST_LrParametr;					//Rezerwa 7	


	lrCapSorterPreScrewerPickerSpeedWhenScrewerShow				:	ST_LrParametr;

END_STRUCT
END_TYPE

// ---- GVLs/GVL.TcGVL
(*
Nazwa:			GVL
Opis:			Zmienne wykorzystywane globalnie
Wersja:			v0.2
Data:			2021-10-05
Autor:			DP,DJ
Urzadzenia:		
Konfiguracja:	
Info:
*)

//{attribute 'qualified_only'}

VAR_GLOBAL
	(******MAIN**********)
	//Ogólne
	bFirstCycle										:BOOL;									// Zmienna pierwszego cyklu
	bManualMode										:BOOL; (**)								// Włączony tryb serwisowy
	tMachineCycleTime								:TIME;									// Czas cyklu maszyny
	bAddGlobalCounter								:BOOL;									// Pomocnicza do dodawania licznika przy odrzucie	
	bAddBadPackageReason							:BOOL;
	bAddBadPackageReason2							:BOOL;
	bChangeover										:BOOL;		
	bPhaseChanging									:BOOL;									// Zmiana trybu na dwufazowy
	bBottleSorterDisable							:BOOL:=FALSE;
	bCapSorterDisable								:BOOL:=FALSE;	
	bFastSpeed										:BOOL;
	
	//Resetowanie 
	bCycleReseting									:BOOL;									//Resetowanie cyklu, trwa 1 sek
	bAllStationDoneDelay							:BOOL;
	bHomingDialog									:BOOL;									//Wyświetl komunikat o bazowaniu
	bHomingCanceled									:BOOL;									// Anulowano bazowanie
	bHoming											:BOOL;									// Trwa bazowanie
	bFirstPositioningDone							:BOOL;
	bRecipeChangePositioning						:BOOL;
	sHomingText										:STRING;
	bResetAfterErrorOrEstop							:BOOL;
	bResetStates									:BOOL;									//Reset cyklu i formatek
	//CycleLogic
	bRobotStationDone								:BOOL;									// Skonczyło się dozowanie lub wyłaczone
	nCheckWeiginhForm								:BOOL;
	//nExitWheelFormsTime							:UINT;									// Czas na wypuszczenie formatki z karuzeli jak pracuje transporter
	
	//Rejestry przesuwne
	bRFIDChecker									:BOOL;									// Sprawdzanie RFID
	bRFIDClearAfterRobot							:BOOL;									// Usuwanie numeru RFID za robotem
	iRFIDClearNr1AfterRobot							:INT;									// Usuwanie numeru RFID za robotem, usuniety = 0
	iRFIDClearNr2AfterRobot							:INT;									// Usuwanie numeru RFID za robotem, usuniety = 0
		
	eClearPackageState								:S_PackageState;
	
	eBottleFeederPackageState						:ARRAY [1..17] OF S_PackageState;		// [1..2] Struktura pod podajnikiem butelek

	eBeforeGatePackageState							:ARRAY [1..17] OF S_PackageState;		// [1..2] Struktura przed szlabane
	eBeforeDispencersPackageState					:ARRAY [1..17] OF S_PackageState;		// [1..4] Struktura przed dozownikami
	eDispencersPackageState							:ARRAY [1..17] OF S_PackageState;		// [1..4] Struktura pod dozownikami
	eAfterDispencersPackageState					:ARRAY [1..17] OF S_PackageState;		// [1..4] Struktura za dozownikami 
	eWeightPackageState								:ARRAY [1..17] OF S_PackageState;		// [1..5] Struktura nad wagami

	eBeforeLidFeeder2PackageState					:ARRAY [1..17] OF S_PackageState;		// [] Struktura przed podawaniem platynek
	eBeforeLidFeederPackageState					:ARRAY [1..17] OF S_PackageState;		// [] Struktura przed podawaniem platynek
	eLidFeederPackageState							:ARRAY [1..17] OF S_PackageState;		// [] Struktura podawania platynek
	eAfterLidFeederPackageState						:ARRAY [1..17] OF S_PackageState;		// [] Struktura przed podawaniem platynek
	eBeforeLidSealerPackageState					:ARRAY [1..17] OF S_PackageState;		// [] Struktura przed zgrzewaniem platynek
	eLidSealerPackageState							:ARRAY [1..17] OF S_PackageState;		// [] Struktura zgrzewanie platynek
	
	eBeforeGateCapSorterPackageState				:ARRAY [1..17] OF S_PackageState;		// [1..4] Struktura przed RFID sortera nasadek
	eBeforeCapSorterPackageState					:ARRAY [1..17] OF S_PackageState;		// [1..4] Struktura przed sorterem
	eCapSorterPackageState							:ARRAY [1..17] OF S_PackageState;		// [1..4] Struktura pod sorterem
	eAfterCapSorterPackageState						:ARRAY [1..17] OF S_PackageState;		// [1..4] Struktura za sorterem
	eBeforeCapControlPackageState					:ARRAY [1..17] OF S_PackageState;		// [1..1] Struktura pod sprawdzaniem obecnosci nakretki
	eBeforeScrewersPackageState						:ARRAY [1..17] OF S_PackageState;		// [1..6] Struktura przed zakręcarkami 
	eBeforeScrewers2PackageState					:ARRAY [1..17] OF S_PackageState;		// [1..6] Struktura przed zakręcarkami przed czujnikiem
	eUnderScrewerPackageState 						:ARRAY [1..17] OF S_PackageState;		// [1..3] Struktura pod zakręcarkami 
	eAfterScrewerPackageState						:ARRAY [1..17] OF S_PackageState;		// [1..8] Struktura za zakręcarkami 
	eUnderCorrectCapPackageState					:ARRAY [1..17] OF S_PackageState;		// [1..7] Struktura pomiedzy robotem a sprawdzeniem poprawnego zakrecenia
	eUnderCorrectCapPackageStateTemp				:ARRAY [1..17] OF S_PackageState;		// [1..7] Struktura pomiedzy robotem a sprawdzeniem poprawnego zakrecenia	
	eRobotPackageState								:ARRAY [1..17] OF S_PackageState;		// [1..2] Struktura pod robotem
	eHistoryPackageState							:ARRAY [1..1000] OF S_PackageState;		// Struktura historyczna przetransferowanych butelek
	eTempState1										:ARRAY [1..17] OF S_PackageState;		// [1..12] Za waga
	eTempState2										:ARRAY [1..17] OF S_PackageState;		// [1..12] Za podajnikiem butelek
	eTempState3										:ARRAY [1..17] OF S_PackageState;		// [1..12] Za sorterem nakretek	
	eRobotTempState									:ARRAY [1..17] OF S_PackageState;    	//  Pod robotem

	// Dodatkowe rejestry przy dozowaniu dwufazowyn
	
	eWeightPackage2PhasePackageState				:ARRAY [1..17] OF S_PackageState;		// [1..5] Struktura nad wagami (** dodane 07.04.2022**)
	eBeforeDispencer34PackageState2Phase			:ARRAY [1..17] OF S_PackageState;		// [1..5] Struktura nad wagami (** dodane 07.04.2022**)
	eDispencer34PackageState2Phase					:ARRAY [1..17] OF S_PackageState;		// [1..5] Struktura nad wagami (** dodane 07.04.2022**)
	eAfterDispencer34PackageState2Phase				:ARRAY [1..17] OF S_PackageState;		// [1..5] Struktura nad wagami (** dodane 07.04.2022**)
	eBeforeDispencer12PackageState2Phase			:ARRAY [1..17] OF S_PackageState;		// [1..5] Struktura nad wagami (** dodane 07.04.2022**)
	eDispencer12PackageState2Phase					:ARRAY [1..17] OF S_PackageState;		// [1..5] Struktura nad wagami (** dodane 07.04.2022**)
	eAfterDispencer12PackageState2Phase				:ARRAY [1..17] OF S_PackageState;		// [1..5] Struktura nad wagami (** dodane 07.04.2022**)

	(******P00_Alarms*****)

	AbActiveWarningDescription								:ARRAY [0..63] OF BOOL;	//  Aktywne ostrzeżenia	
	
	//Sygnał dzwiekowy
	bSoftAlarm										:BOOL;
	
	bResetError										:BOOL:=FALSE;(**)						// Zmienna resetująca stację/błąd w PLC ,wystawia się po wciśnięciu ResetVisuCmd			
	//Reset Diagnostyki	
	
	//Alarmy inne*
	GeneralAlarms									:S_Error;								// 1 Ogólne
	//*Alarmy Stacji
	FormTransporterDispencerError					:S_Error;								// 2 Transporter wwjazdowy pod dozowniki
	FormTransporterScrewerError						:S_Error;								// 2 Transporter wyjściowy
	FormTransporterROPPError						:S_Error;
	FormTransporterAfterCapSorterError				:S_Error;
	FormTransporterBeforeScrewerError				:S_Error; 								// 3 Transporrter przed zakręcarkami
	FormTransporterSlowerError						:S_Error; 								// Spowalniacz
	FormTransporterAfterScrewerError				:S_Error; 								// 3 Transporrter przed zakręcarkami
	FormTransporterAfterBottleTransferError			:S_Error; 								
	BottleFeederError								:S_Error;								// Podajnik butelek
	BottleFeederTurnTableError						:S_Error;								// Stół obrotowy podajnika butleek
	BottleFeederFormGateError						:S_Error;								// Stoper formatek
	PucksInserterError								:S_Error;								// Podajnik butelek
	PucksInserterTurnTableError						:S_Error;								// Stół obrotowy podajnika opakowań
	PucksInserterFormGateError						:S_Error;								// Stoper formatek
	PucksInserterPushTableError_m1					:S_Error;								//71U3
	PucksInserterPushTableError_m2					:S_Error;								//71U4
	PucksInserterPushTableError_m3					:S_Error;								//
	GateBeforeDispencersError						:S_Error;		   						// 3A Szlaban przed dozownikami
		

	BarrierBetweenDispencers						:S_Error;								// Obsługa błędów szlaban dozowniki ( dozowanie dwufazowe, pod dozownikamia);
	BarrierBetweenWeights							:S_Error;								// Obsługa błędów stacji szlabanu pomiedzy wagamia ( dozowanie dwufazowe, wjazd na wagi);
	
	// Alarm wyciągu
	
	ExhaustFanError									:S_Error;
	SensorAcetoneError								:S_Error;								// Obśługa błedów czujnika acetonu
	SensorAirFlowError								:S_Error;								// Obsługa błędów czujnika przepływu 
	
	BottlePusherError								:S_Error;	
	//DispencerGatesError							:S_Error;								// 4 Szlabany pod dozownikami
	DispencersDragLeftError							:S_Error;								// Przeciąganie formatek
	DispencersDragRightError						:S_Error;								// Przeciąganie formatek (** 15.04.22 Damian**)
	

	DispencersCatch1Error							:S_Error;								// 4 Chwytak butelek dozownika 1
	DispencersCatch2Error							:S_Error;								// 4 Chwytak butelek dozownika 2
	DispencersCatch3Error							:S_Error;								// 4 Chwytak butelek dozownika 3
	DispencersCatch4Error							:S_Error;								// 4 Chwytak butelek dozownika 4
	Dispencer1Error									:S_Error;								// 5 Dozownik nr 1
	Dispencer2Error									:S_Error;								// 6 Dozownik nr 2
	Dispencer3Error									:S_Error;								// 6 Dozownik nr 3	
	Dispencer4Error									:S_Error;								// 6 Dozownik nr 4		
	TankHeatingError								:S_Error;								// Grzanie zbiornka

	WeightLiftError									:S_Error;
	
	Weight1Error									:S_Error;								// 8 Waga pierwsza jednofazowe
	Weight2Error									:S_Error;								// 8 Waga druga jednofazowe
	Weight3Error									:S_Error;								// 8 Waga trzecia jednofazowe
	Weight4Error									:S_Error;								// 8 Waga czwarta jednofazowe
	Weight5Error									:S_Error;								// 8 Waga piąta jednofazowe   	(** dodane 07.04.2022**)
	Weight6Error									:S_Error;								// 8 Waga szósta jednofazowe	(** dodane 07.04.2022**)
	
	
	GateAfterWeightError							:S_Error;								// 9 Szlaban za wagamia
		
	Dispencer1CorrectionError						:S_Error;	
	Dispencer2CorrectionError						:S_Error;
	Dispencer3CorrectionError						:S_Error;	
	Dispencer4CorrectionError						:S_Error;	
	WickFeederSorterError							:S_Error;
	
	
	CapFeederError									:S_Error;								// 14 
	CapSorterDragError								:S_Error;								// 15  Przeciąganie pod sorterem nasadek
			
	CapPuttedCheckError								:S_Error;								// 17 Wykrycie zakrętki
	
	GripperScrewerCatch1Error						:S_Error;								// 18 Chwytak zakręcarki szczękowej
	GripperScrewerCatch2Error						:S_Error;								// 18 Chwytak zakręcarki szczękowej
	GripperScrewer1Error							:S_Error;								// 19 Zakręcerka szczękowa 1
	GripperScrewer2Error							:S_Error;								// 19 Zakręcerka szczękowa 1

	BottleDragError									:S_Error;								//19.1 Przeciąganie butelek pod zakręcarkami
	CapCorrectCheckError							:S_Error;								// 21B Sprawdzanie zakręconej nakrętki
	CapCorrectCheckCameraError						:S_Error;
	BottleTransferError								:S_Error;								// 22 Robot
	GateRobotError									:S_Error;								// 22 Szlabany pod robotem
	BottleTransferAfterDragError					:S_Error;								// 14 

	BadBottleConveyorError							:S_Error;								// 23 Transporter odrzuconych butelek	
	LabelMachineError								:S_Error;								// 24 Etykieciarka
	TanksError										:S_Error;								// 24 Zbiorniki
	ExitTurnTableError								:S_Error;								// 25 Stół odbierający
	ExitConveyorError								:S_Error;								// 


	BarrierLidFeeder								: S_Error;								// Podajnik platynek 
	LidFeederError									: S_Error;								// Podajnik platynek 
	LidFeeder2Error									: S_Error;								// Podajnik platynek 2
	LidFeederFormPositioningError					: S_Error;	
						
	BarrierWickFeeder								: S_Error;
	WickFeederDragError								: S_Error;
	WickFeederError									: S_Error;
	WickFeeder2Error								: S_Error;
	WickFeederFormPositioningError					: S_Error;
	
	LidFeederDragError								: S_Error;								// Przeciąganie formatek                                                                                          
	LidPuttedCheckError								: S_Error;								// Wykrycie platynki                                                                                         
	LidSealerError									: S_Error;								// Zgrzewarka 1
	LidSealer2Error									: S_Error;								// Zgrzewarka 2
	LidSealerDragError								: S_Error;								// Przeciąganie formatek
	
	
	
	
	//Warningi
	TanksWarning									:ARRAY [0..7] OF S_Warning;							
	BottleTransferWarning							:ARRAY [0..7] OF S_Warning;	
	GeneralWarning1									:ARRAY [0..7] OF S_Warning;
	WeightWarning									:ARRAY [0..7] OF S_Warning;		
	DispencersWarning								:ARRAY [0..7] OF S_Warning;		
	ScrewersWarning									:ARRAY [0..7] OF S_Warning;		
	BottleFeederWarning								:ARRAY [0..7] OF S_Warning;
	ExSensorWarning									:ARRAY [0..7] OF S_Warning;
	CapFeederWarning								:ARRAY [0..7] OF S_Warning;	
	CapSorterWarning								:ARRAY [0..7] OF S_Warning;		
	BottleSorterWarning								:ARRAY [0..7] OF S_Warning;	
	LidFeederWarning								:ARRAY [0..7] OF S_Warning;		
	WickFeederWarning								:ARRAY [0..7] OF S_Warning;	
	WickFeederSorterWarning							:ARRAY [0..7] OF S_Warning;	
	(********P00_OEE********)		
	udiCounterExecuteTimeTemp						:UDINT;
	udiCounterErrorTimeTemp							:UDINT;
	udiCounterReadyTimeTemp							:UDINT;

	
	(******P00_Basic*******)
	//impulsy
	bImp1Sec										:BOOL;									// Impuls na zbocze generatora 1 sek
	b1Hz											:BOOL;									// Generator 1 sekundowy
	bV1Hz											:BOOL;									// bit o czest. 1Hz
	b2Hz											:BOOL;									// Generator 0,5 sekundowy
	//czas
	dtActTime										:DT;
	wYear 											:WORD;
	wMonth											:WORD;
	wDayOfWeek 										:WORD;
	wDay 											:WORD;
	wHour 											:WORD;
	wMinute 										:WORD;
	wSecond 										:WORD;
	wMilliseconds 									:WORD;

	//Zmienne podst.
	bAlwaysFalse									:BOOL:=FALSE;							//Zawsze zero
	
	(*****P00_PneumaticsValves***)
	(*****Receptury****)	
	bVTEMEnable										:BOOL;
	lrGripperScrewerPressure						:LREAL;									//Ciśnienie siłownika chwytaka nasadki zakręcarki szczękowej 1 (0.0 kg)
	lrGripperScrewerPressureExhaustLevel			:LREAL;									//Prędkość zamykania siłownika chwytaka nasadki zakręcarki szczękowej 1 (0.0-100.0 %)
	lrGripperScrewerCatchPressure					:LREAL;									//Ciśnienie siłownika chwytaka butelki zakręcarki szczękowej 1 (0.0 kg)
	lrGripperScrewerCatchPressureExhaustLevel		:LREAL;									//Prędkość zamykania siłownika chwytaka butelki zakręcarki szczękowej 1 (0.0-100.0 %)
	lrDispencerCatchPressure						:LREAL;

	(*****P0_Recipes***)
	(*****Receptury****)
	sRecipeName										:STRING;				
	sRecipeIndex									:STRING;				
	nRecipeIndex									:REAL;					
	bRecipeAfterPowerStateChosen					:BOOL;									//Receptura w stanie Power została wybrana (Pierwsza receptura po uruchomieniu)
	iPackageCapType									:INT; 									// Typ nasadki 
	iPackageCapDiameter								:INT;
	
	//[H] Praca w trybie wybuchowym
	bExEnable										:BOOL;						// [H] Tryb EX
	
	
	(****P01_BottleFeeder****)
	bBottleFeederEnable								:BOOL;									// Zezwolenie na pracę stacji podawania opakowań
	bBottleFeederDoHoming							:BOOL;									// Wykonanie bazowania stacji podawania butelek
	bBottleFeederTurnTableRun						:BOOL;									// Komenda startu stołu obrotwego
	iBottleFeederBottleSensorDelay					:INT;
	iBottleFeederFormGateDelay						:INT;
	iBottleFeederAllowFormDelay						:INT;
	bBottleFeederFormGateRun						:BOOL;									// Bit sterujacy działanie bramki 
	iBottleFeederTurntableVelocitySV				:UDINT;	

	(****P01_PucksInserter****)
	bPucksInserterEnable							:BOOL;									// Zezwolenie na pracę stacji 
	bPucksInserterDoHoming							:BOOL;									// Wykonanie bazowania stacji 
	bPucksInserterTurnTableRun						:BOOL;									// Komenda startu stołu obrotwego
	iPucksInserterBottleSensorDelay					:INT;
	iPucksInserterFormGateDelay						:INT;
	iPucksInserterFormGateDelayAdd					:INT;	
	iPucksInserterAllowFormDelay					:INT;
	bPucksInserterFormGateRun						:BOOL;									// Bit sterujacy działanie bramki 
	iPucksInserterTurntableVelocitySV				:UDINT;	
	iPucksInserterConveyorVelocitySV				:UDINT;	
	aPucksInserterWheelAxisRef						:AXIS_REF;								// Struktura osi 
	lrPucksInserterWheelOffset						:LREAL;									// Offset karuzeli +-10 st.
	lrPucksInserterWheelAcceleration				:LREAL;									// Przyspieszenie 
	lrPucksInserterWheelVelocity					:LREAL;									// Prędkość 
	lrPucksInserterHammerHeightSV					:LREAL;									// Pozycja
	
	//Push table 27.05 Vasyl	
	bPucksInserterPushTable_m1_Enable					:BOOL;
	bPucksInserterPushTable_m1_Run						:BOOL;
	udiPucksInserterPushTable_m1_VelocitySV				:UDINT;
	bPucksInserterPushTable_m2_Enable					:BOOL;
	bPucksInserterPushTable_m2_Run						:BOOL;
	udiPucksInserterPushTable_m2_VelocitySV				:UDINT;
	bPucksInserterPushTable_m3_Enable					:BOOL;
	bPucksInserterPushTable_m3_Run						:BOOL;
	udiPucksInserterPushTable_m3_VelocitySV				:UDINT;

	udiPucksInserterPushTableActuatorPUSHDelay			:UDINT;
	udiPucksInserterPushTableActuatorPULLDelay			:UDINT;
	udiPucksInserterPushTableOFFDelay					:UDINT;

	(****P01_BottleSorter****)
	//Po komunikacji
	
	(*****P01_Gates********)
	bGateBeforeDispencersEnable						:BOOL;									//Zezwolenie na pracę szlabanów pod robotem
	nGateBeforeDispencersTimeFormInserting			:UINT;									//Czas od momentu wjazdu formatek do zamkniecia 1 szlabanu pod robotem
	
	bGateAfterWeightEnable							:BOOL;									//Zezwolenie na pracę szlabanów pod robotem
	nGateAfterWeightTimeFormInserting				:UINT;									//Czas od momentu wjazdu formatek do zamkniecia 1 szlabanu pod robotem
		
	bBarrierLidFeederEnable							:BOOL;									//Zezwolenie na pracę szlabanów pod robotem
	nBarrierLidFeederTimeFormInserting				:UINT;									//Czas od momentu wjazdu formatek do zamkniecia 1 szlabanu pod robotem
	
	bGateRobotEnable								:BOOL;									//Zezwolenie na pracę szlabanów pod robotem
	nGateRobotTimeFormInserting						:UINT;									//Czas od momentu wjazdu formatek do zamkniecia 1 szlabanu pod robotem
	
	(*****P01_Barriers********)
	bBarrierWeightRun								:BOOL;									// Komenda otwarcia bariery przed wagami
	bBarrierDispencerRun							:BOOL;									// Komenda otwarcia bariery przed wagami
	
	(*****P02_Dispencers***)
	bCIP											: BOOL; // Włączone mycie CIP
	bDispencer1Cleaning								: BOOL;	// Mycie dozowników
	bDispencer2Cleaning								: BOOL;	// Mycie dozowników
	bDispencer3Cleaning								: BOOL;	// Mycie dozowników
	bDispencer4Cleaning								: BOOL;	// Mycie dozowników

	bDispencer1DoSync								: BOOL;	// Ustawienie tłoka/podnośnika 1 dozownika na konkretną pozycję (otwierają się zawory ssania) tylko w trybie serwisowym 
	bDispencer2DoSync								: BOOL;	// Ustawienie tłoka/podnośnika 2 dozownika na konkretną pozycję (otwierają się zawory ssania) tylko w trybie serwisowym 
	bDispencer3DoSync								: BOOL;	// Ustawienie tłoka/podnośnika 3 dozownika na konkretną pozycję (otwierają się zawory ssania) tylko w trybie serwisowym 
	bDispencer4DoSync								: BOOL;	// Ustawienie tłoka/podnośnika 4 dozownika na konkretną pozycję (otwierają się zawory ssania) tylko w trybie serwisowym 

	//Dozowniki 
	bDispencer12AllowDosingAfterDrag				:BOOL;
	bDispencer34AllowDosingAfterDrag				:BOOL;	
	bDoorDispencerOpen								:BOOL;
	bDosingTwoPhases								:BOOL;									//Dozowanie dwu fazowe
	bDispencersDoHoming								:BOOL;									//Wykonanie bazowania dozowniki
    lrDispencersLifterReadyPosition					:LREAL;									//Pozycja podnonika przy której dozowniki są w stanie gotowości
	uiDispencerStartDosingDelay						:UINT;(*0-3000*)				 		// Czas opóźnienia rozpoczęcia dozowania

//	Dozownik 1
	aDispencer1AxisRef								:AXIS_REF;//ActPos	(**)				// Struktura osi dozownika 1
	aDispencerLifter12AxisRef						:AXIS_REF;//ActPos	(**)				// Struktura osi dozownika 1
	bDispencer1Enable								:BOOL; 									// Zezwolenie na prace dozownika 1
	lrDispencer1DoseVolume							:LREAL:=195; 							// Objętoć do wydozowania przez dozownik 1
	bDispencer1LiftSynchroPh1						:BOOL;						 			// Polecenie synchronizacji dozownika z podnonikiem w fazie 1 Dozownika 1
	bDispencer1LiftSynchroPh2						:BOOL; 					 				// Polecenie synchronizacji dozownika z podnonikiem w fazie 2 Dozownika 1
	bDispencer1LiftSynchroPh3						:BOOL; 									// Polecenie synchronizacji dozownika z podnonikiem w fazie 3 Dozownika 1
	lrDispencer1Phase1Volume						:LREAL:=100;							// Objętoć do której ma trwać faza pierwsza dozowania dozownika 1
	lrDispencer1Phase2Volume						:LREAL:=100;							// Objętoć do której ma trwać faza druga dozowania dozownika 1
	lrDispencer1Phase1Velocity						:LREAL:=500;							// Prędkoć z jakš ma byc wykonywana faza pierwsza dozowania dozownika 1
	lrDispencer1Phase2Velocity						:LREAL:=500;							// Prędkoć z jakš ma byc wykonywana faza druga dozowania dozownika 1
	lrDispencer1Phase3Velocity						:LREAL:=500;							// Prędkoć z jakš ma byc wykonywana faza trzecia dozowania dozownika 1
	lrDispencer1SuckVelocity						:LREAL:=500;							// Prędkoć z jakš ma byc wykonywane zasysanie dozownika 1
	lrDispencer1Phase1Acceleration					:LREAL:=3000;							// Przyspieszenie z jakim ma byc wykonywana faza 1  dozownika 1
	lrDispencer1Phase2Acceleration					:LREAL:=3000;							// Przyspieszenie z jakim ma byc wykonywana faza 2  dozownika 1
	lrDispencer1Phase3Acceleration					:LREAL:=3000;							// Przyspieszenie z jakim ma byc wykonywana faza 3  dozownika 1
	lrDispencer1SuckAcceleration					:LREAL:=3000;							// Przyspieszenie z jakim ma byc wykonywane zasysanie dozownika 1
	lrDispencer1Phase1Deceleration					:LREAL:=3000;							// Zwalnianie z jakim ma byc wykonywana faza 1  dozownika 1
	lrDispencer1Phase2Deceleration					:LREAL:=3000;							// Zwalnianie z jakim ma byc wykonywana faza 2  dozownika 1
	lrDispencer1Phase3Deceleration					:LREAL:=3000;							// Zwalnianie z jakim ma byc wykonywana faza 3  dozownika 1
	udiDispencer1DosingDoneDelayTime				:UDINT:=20; 							// Opóźnienie wykonania cyklu dozy przez dozownik 1 [ms]
	lrDispencer1SuckValveOpenVolume					:LREAL:=0;(*Z 0-15*)					//[3] Objętość przy której ma byc otwierany zawór ssania dozownika 1
	lrDispencer1SuckValveOpenTimeDelay				:LREAL:=0;(*NOWA 0-1000*)				// [3] Opóżnienie rozpoczęcia ssania po tłoczeniu [ms]
	lrDispencer1SuckValveCloseVolume				:LREAL:=0;(*Z 0-15*)					// [4] Objętość przy której ma byc zamykany zawór ssania dozownika 1
	lrDispencer1SuckValveCloseTimeDelay				:LREAL:=0;(*NOWA 0-2000*)				// [4] Opóżnienie zamknięcia zaworu ssącego [ms]
	lrDispencer1DoseValveOpenVolume					:LREAL:=0;(*Z 0-15*)					//[1] Objętość przy której ma byc otwierany zawór tłoczenia (iglica) dozownika 1 
	lrDispencer1DoseValveOpenTimeAcc				:LREAL:=0;(*NOWA 0-500*)				// [1] Przyśpieszenie otwarcia zaworu tłoczenia [ms]
	lrDispencer1DoseValveCloseVolume				:LREAL:=0;(*0-15*)						// [2] Objętość przy której ma byc zamykany zawór tłoczenia (iglica) dozownika 1 
	lrDispencer1DoseValveCloseTimeDec				:LREAL:=0;(*NOWA 0-1000*)				// [2] Opóźnienie zamknięcia zaworu tłoczenia [ms]
	lrDispencer1DoseSuckingVolume					:LREAL:=0;(*NOWA 0-100*)			  	//[5] [Podsysanie] Wartość dozy do posysenia [ml]	
	lrDispencer1DoseSuckingTimeDelay				:LREAL:=0;(*NOWA 0-500*)  				//[6] [Podsysanie] Opóźnienie podsysania [ms]
	bDispencer1DoseSucking							:BOOL;(*NOWA*) 					 		// [Podsysanie] Opcja podsysania przy dozowaniu
	lrDispencer1LifterStartDosePosition				:LREAL:=20;								// Pozycja podnonika przy której rozpoczyna sie dozowanie dozownika 1
	lrDispencer1LifterStopDosePosition				:LREAL:=60;								// Pozycja podnonika przy której kończy sie dozowanie dozownika 1
	lrDispencer1LifterVelocity						:LREAL:=20;								// Prędkoć podnonika dozownika 1	
	lrDispencer1LifterAcceleration					:LREAL:=2;								// Przyspieszenie podnonika dozownika 1
	lrDispencer1LifterDeceleration					:LREAL:=2;								// Przyspieszenie podnonika dozownika 1

//	Dozownik 2
	aDispencer2AxisRef								:AXIS_REF;//ActPos(**)					// Struktura osi dozownika 2
	bDispencer2Enable								:BOOL; 									// Zezwolenie na prace dozownika 2
	lrDispencer2DoseVolume							:LREAL:=195; 							// Objętoć do wydozowania przez dozownik 2
	bDispencer2LiftSynchroPh1						:BOOL;						 			// Polecenie synchronizacji dozownika z podnonikiem w fazie 1 Dozownika 2
	bDispencer2LiftSynchroPh2						:BOOL; 					 				// Polecenie synchronizacji dozownika z podnonikiem w fazie 2 Dozownika 2
	bDispencer2LiftSynchroPh3						:BOOL; 									// Polecenie synchronizacji dozownika z podnonikiem w fazie 3 Dozownika 2
	lrDispencer2Phase1Volume						:LREAL:=100;							// Objętoć do której ma trwać faza pierwsza dozowania dozownika 2
	lrDispencer2Phase2Volume						:LREAL:=100;							// Objętoć do której ma trwać faza druga dozowania dozownika 2
	lrDispencer2Phase1Velocity						:LREAL:=500;							// Prędkoć z jakš ma byc wykonywana faza pierwsza dozowania dozownika 2
	lrDispencer2Phase2Velocity						:LREAL:=500;							// Prędkoć z jakš ma byc wykonywana faza druga dozowania dozownika 2
	lrDispencer2Phase3Velocity						:LREAL:=500;							// Prędkoć z jakš ma byc wykonywana faza trzecia dozowania dozownika 2
	lrDispencer2SuckVelocity						:LREAL:=500;							// Prędkoć z jakš ma byc wykonywane zasysanie dozownika 2
	lrDispencer2Phase1Acceleration					:LREAL:=3000;							// Przyspieszenie z jakim ma byc wykonywana faza 1  dozownika 2
	lrDispencer2Phase2Acceleration					:LREAL:=3000;							// Przyspieszenie z jakim ma byc wykonywana faza 2  dozownika 2
	lrDispencer2Phase3Acceleration					:LREAL:=3000;							// Przyspieszenie z jakim ma byc wykonywana faza 3  dozownika 2
	lrDispencer2SuckAcceleration					:LREAL:=3000;							// Przyspieszenie z jakim ma byc wykonywane zasysanie dozownika 2
	lrDispencer2Phase1Deceleration					:LREAL:=3000;							// Zwalnianie z jakim ma byc wykonywana faza 1  dozownika 2
	lrDispencer2Phase2Deceleration					:LREAL:=3000;							// Zwalnianie z jakim ma byc wykonywana faza 2  dozownika 2
	lrDispencer2Phase3Deceleration					:LREAL:=3000;							// Zwalnianie z jakim ma byc wykonywana faza 3  dozownika 2
	udiDispencer2DosingDoneDelayTime				:UDINT:=20; 							// Opóźnienie wykonania cyklu dozy przez dozownik 2 [ms]
	lrDispencer2SuckValveOpenVolume					:LREAL:=0;(*Z 0-15*)					// [3] Objętość przy której ma byc otwierany zawór ssania dozownika 2
	lrDispencer2SuckValveOpenTimeDelay				:LREAL:=0;(*NOWA 0-1000*)				// [3] Opóżnienie rozpoczęcia ssania po tłoczeniu [ms]
	lrDispencer2SuckValveCloseVolume				:LREAL:=0;(*Z 0-15*)					// [4] Objętość przy której ma byc zamykany zawór ssania dozownika 2
	lrDispencer2SuckValveCloseTimeDelay				:LREAL:=0;(*NOWA 0-2000*)				// [4] Opóżnienie zamknięcia zaworu ssącego [ms]
	lrDispencer2DoseValveOpenVolume					:LREAL:=0;(*Z 0-15*)					// [1] Objętość przy której ma byc otwierany zawór tłoczenia (iglica) dozownika 2 
	lrDispencer2DoseValveOpenTimeAcc				:LREAL:=0;(*NOWA 0-500*)				// [1] Przyśpieszenie otwarcia zaworu tłoczenia [ms]
	lrDispencer2DoseValveCloseVolume				:LREAL:=0;(*0-15*)						// [2] Objętość przy której ma byc zamykany zawór tłoczenia (iglica) dozownika 2 
	lrDispencer2DoseValveCloseTimeDec				:LREAL:=0;(*NOWA 0-1000*)				// [2] Opóźnienie zamknięcia zaworu tłoczenia [ms]
	lrDispencer2DoseSuckingVolume					:LREAL:=0;(*NOWA 0-100*)  				// [5] [Podsysanie] Wartość dozy do posysenia [ml]	
	lrDispencer2DoseSuckingTimeDelay				:LREAL:=0;(*NOWA 0-500*)  				// [6] [Podsysanie] Opóźnienie podsysania [ms]
	bDispencer2DoseSucking							:BOOL;(*NOWA*)  						// [Podsysanie] Opcja podsysania przy dozowaniu
	lrDispencer2LifterStartDosePosition				:LREAL:=20;								// Pozycja podnonika przy której rozpoczyna sie dozowanie dozownika 2
	lrDispencer2LifterStopDosePosition				:LREAL:=60;								// Pozycja podnonika przy której kończy sie dozowanie dozownika 2
	lrDispencer2LifterVelocity						:LREAL:=20;								// Prędkoć podnonika dozownika 2	
	lrDispencer2LifterAcceleration					:LREAL:=2;								// Przyspieszenie podnonika dozownika 2
	lrDispencer2LifterDeceleration					:LREAL:=2;								// Przyspieszenie podnonika dozownika 2

	//	Dozownik 3
	aDispencer3AxisRef								:AXIS_REF;//ActPos	(**)				// Struktura osi dozownika 3
	aDispencerLifter34AxisRef						:AXIS_REF;//ActPos	(**)				// Struktura osi dozownika 3
	bDispencer3Enable								:BOOL; 									// Zezwolenie na prace dozownika 3								

	//	Dozownik 4
	aDispencer4AxisRef								:AXIS_REF;//ActPos				(**)	// Struktura osi dozownika 4
	bDispencer4Enable								:BOOL; 									// Zezwolenie na prace dozownika 4
		
	//Podonosnik chwytaka i tacki 1,2,3,4
	bDispencersCatchEnable								:BOOL; 									// Zezwolenie na pracę chwytaka butelek pod dozownikami 1
	bDispencersCatchMaxPressure							:BOOL;									// Zwiekszona siła chwytania
	bDispencersCatch1DoHoming							:BOOL;									// Wykonanie bazowania przez chwytak i tacke pod dozownikiem 1
	lrDispencersCatchHeightSV							:LREAL:=36;  					       	// Zadana wartoć pozycji bazowania stacji chwytania opakowania pod dozownikami
	bDispencersCatch2DoHoming							:BOOL;									// Wykonanie bazowania przez chwytak i tacke pod dozownikiem 2
	bDispencersCatch3DoHoming							:BOOL;									// Wykonanie bazowania przez chwytak i tacke pod dozownikiem 3
	bDispencersCatch4DoHoming							:BOOL;									// Wykonanie bazowania przez chwytak i tacke pod dozownikiem 4

    (*Wartości dla nowych czujników wykrywania butelki pod dozownikami*)
    (*Są zależne od szerokości szyjki i dlatego trzeba je zapamiętywać*)
    (*Kalibracja chwytaków w serwisie będzie nadpisywała te wartości*)
    (*Będzie się je zmieniało przez kalibracje więc widocznośc tylko ustawić dla serwisu*)
    lrDispencersCatch1ClosedValue                    	:LREAL;                        // Chwytak 1 | wartość kalibracji zamkniętego chwytaka
    lrDispencersCatch1OpenValue                      	:LREAL;                        // Chwytak 1 | wartość kalibracji otwartego chwytaka
    lrDispencersCatch2ClosedValue                    	:LREAL;                        // Chwytak 2 | wartość kalibracji zamkniętego chwytaka
    lrDispencersCatch2OpenValue                      	:LREAL;                        // Chwytak 2 | wartość kalibracji otwartego chwytaka
    lrDispencersCatch3ClosedValue                   	:LREAL;                        // Chwytak 3 | wartość kalibracji zamkniętego chwytaka
    lrDispencersCatch3OpenValue                     	:LREAL;                        // Chwytak 3 | wartość kalibracji otwartego chwytaka
    lrDispencersCatch4ClosedValue                   	:LREAL;                        // Chwytak 4 | wartość kalibracji zamkniętego chwytaka
    lrDispencersCatch4OpenValue                      	:LREAL;                        // Chwytak 4 | wartość kalibracji otwartego chwytaka
    (*Tolerancja dla chwytaków - dla operatora*)
    lrDispencersCatchTolerance                       	:LREAL;                        // Tolerancja szyjki butelki pod dozownikami [0-100%]      
	
	//Przeciąganie formatek
	aFormsDragingRightAxisRef							:AXIS_REF;								// Struktura osi napędu krokowego przeciągania	
	bFormsDragingRightEnable							:BOOL;									// Zezwolenie na pracę przeciągania 
	bFormsDragingRightDoHoming							:BOOL;									// Wykonanie bazowania przeciągania
	bFormsDragingRightHeightSet							:BOOL;									// Wykonanie bazowania przeciągania
	lrFormsDragingRightVelocity							:LREAL:=100;							// Prędkośc przeciągania
	lrFormsDragingRightAcceleration						:LREAL:=12;								// Przyspieszenie przeciągania
	lrFormsDragingRightDeceleration						:LREAL:=15;								// Hamowanie przeciągania
	bFormsDragingRightPrepareRun						:BOOL;
	bFormsDragingRightRunCheck							:BOOL;		
	//Przeciąganie formatek
	aFormsDragingLeftAxisRef							:AXIS_REF;								// Struktura osi napędu krokowego przeciągania
	bFormsDragingLeftEnable								:BOOL;									// Zezwolenie na pracę przeciągania 
	bFormsDragingLeftDoHoming							:BOOL;									// Wykonanie bazowania przeciągania
	bFormsDragingLeftHeightSet							:BOOL;									// Wykonanie bazowania przeciągania
	lrFormsDragingLeftVelocity							:LREAL:=100;							// Prędkośc przeciągania
	lrFormsDragingLeftAcceleration						:LREAL:=12;								// Przyspieszenie przeciągania
	lrFormsDragingLeftDeceleration						:LREAL:=15;								// Hamowanie przeciągania
	bFormsDragingLeftPrepareRun							:BOOL;
	iFormsDragingFormCounter							:INT;
	bFormsDragingLeftRunCheck							:BOOL;	
	
	//Zbiorniki
	bTank1MixerEnable								:BOOL;(**)   					  		// Załaczanie mieszadła zbiornikowego 1
	bTankHeatingEnable								:BOOL;								    // Zezwolenie na pracę
	iTankHeatingTempSV								:INT;	
	bTank1SupplyPumpEnable							:BOOL;(**) 								// Załaczanie pompy zasilajacej zbiornik 1
	bTank1PressureEnable							:BOOL;									// Włączanie Ciśnienia w zbiorniku 1
	bTank2SupplyPumpEnable							:BOOL;(**) 								// Załaczanie pompy zasilajacej zbiornik 2
	uTank1LevelSetpoint								:UINT;(*o*)								// Wartość zadana masy do czujnika poziomu w zbiorniku nr 1
	bTank1LevelSignalInvert							:BOOL;									// Odwróć sygnał z czujnika zbiornika pierwszego
	bTank2LevelSignalInvert							:BOOL;									// Odwróć sygnał z czujnika zbionirka drugiego
	uTank2LevelSetpoint								:UINT;(*o*)								// Wartość zadana masy do czujnika poziomu w zbiorniku nr 1
	//Zbiorniki-dodatkowe
	bTankRainbowMode								:BOOL;
	(*****P05_Weight*****)
	bWeightLiftEnable								:BOOL;	
	bWeightLiftDoHoming								:BOOL;
	bWeightLiftDeparture							:BOOL;
	bWeight1234ReleaseBlock							:BOOL;	
	bWeightLift2PhaseRun							:BOOL;
	bWeight56ReleaseBlock							:BOOL;	
	bWeighingAutoTarePreset							:BOOL;	
	bWeighingAutoTare								:BOOL;	
	
	bWeight1Enable									:BOOL;									// Zezwolenie na pracę wagi 1
	lrWeightMassSV									:LREAL;									// Waga zadana masy 
	lrWeight1Chart									:LREAL;									// Tylko do wykresów
	lrWeight2Chart									:LREAL;									// Tylko do wykresów
	lrWeight3Chart									:LREAL;									// Tylko do wykresów
	lrWeight4Chart									:LREAL;									// Tylko do wykresów
	lrWeight5Chart									:LREAL;									// Tylko do wykresów
	lrWeight6Chart									:LREAL;									// Tylko do wykresów
	
	iWeight1ActuatorUpDelay							:INT;									// Opóźnienie podnoszenia Waga 1	
	iWeight2ActuatorUpDelay							:INT;									// Opóźnienie podnoszenia Waga 2	
	iWeight3ActuatorUpDelay							:INT;									// Opóźnienie podnoszenia Waga 3	
	iWeight4ActuatorUpDelay							:INT;									// Opóźnienie podnoszenia Waga 4	
	iWeight5ActuatorUpDelay							:INT;									// Opóźnienie podnoszenia Waga 5	
	iWeight6ActuatorUpDelay							:INT;									// Opóźnienie podnoszenia Waga 6	
	iWeight56ActuatorUpAddDelay						:INT;									// Opóźnienie podnoszenia Waga 5	
	iWeight14ActuatorUpAddDelay						:INT;									// Opóźnienie podnoszenia Waga 5	

	//Podajnik knotów
	bWickFeederEnable								: BOOL;									// Zezwolenie na pracę podajnika platynek
	bWickFeederDoHoming								: BOOL;									// Bazowanie podajnika platynek
   lrWickFeederHeightPosSV							: LREAL := 72;							// Wysokoć na której ma znajdować się podajnik platynek

	//Przeciąganie podajnik knotów
	bWickFeederDragingStationEnable					: BOOL;
	bWickFeederDragingStationDoHoming				: BOOL;
	bWickFeederDragingStationPrepareRun				: BOOL;
	lrWickFeederDragingStationVelocity				: LREAL; 							// Zadana prędkosć ruchu przeciągania formatek pod zakręcarkam
	lrWickFeederDragingStationAcceleration			: LREAL;							// Przyspieszenie przeciągania
	lrWickFeederDragingStationDeceleration			: LREAL;							// Hamowanie przeciągania
	aWickFeederDragingAxisRef						: AXIS_REF;
	bWickFeederDragingHeightSet						: BOOL;	
	iWickFeederSorterTimeDelayOn					: INT;
	iWickFeederSorterTimeDelayOff					: INT;
	iWickFeederSorterTimeToEmptySleeveError			: INT;

	//Podajnik platynek
	bLidFeederEnable								: BOOL;									// Zezwolenie na pracę podajnika platynek
	bLidFeederDoHoming								: BOOL;									// Bazowanie podajnika platynek
    bLidFeederHeaterEnable							: BOOL;									// Zezwolenie na prace grzałki podajnika platynek
	iLidFeederHeatingTime							: INT 	:= 1000;						// Czas zgrzewania wstępnego podajnika platynek [ms]
    lrLidFeederHeightPosSV							: LREAL := 72;							// Wysokoć na której ma znajdować się podajnik platynek
    iLidFeeder1TempSV								: INT	:= 150;							// Temperatura zadana grzałki podajnika platynek
    iLidFeeder2TempSV								: INT	:= 150;							// Temperatura zadana grzałki podajnika platynek
	iLidFeederTempHisteresis						: INT;							 	  	// Histereza poprawnej temperatury grzałki (+/- *C), po jej przekroczeniu grzałka wpada w błšd
	bLidFeeder2Enable								: BOOL;									// Zezwolenie na pracę podajnika platynek	
	bLidFeederFormPositioningRun					: BOOL;	
	
	//Przeciąganie podajnik platynek
	bLidFeederDragingStationEnable					: BOOL;
	bLidFeederDragingStationDoHoming				: BOOL;
	bLidFeederDragingStationPrepareRun				: BOOL;
	lrLidFeederDragingStationVelocity				: LREAL; 							// Zadana prędkosć ruchu przeciągania formatek pod zakręcarkam
	lrLidFeederDragingStationAcceleration			: LREAL;							// Przyspieszenie przeciągania
	lrLidFeederDragingStationDeceleration			: LREAL;							// Hamowanie przeciągania
	aLidFeederDragingAxisRef						: AXIS_REF;
	bLidFeederDragingHeightSet						: BOOL;		                                                											
 													
	//Sprawdzanie platynek                          
   	bLidPuttedCheckDoHoming     					: BOOL;  								// Wykonanie bazowania stacji sprawdzania nakrętek
    bLidPuttedCheckEnable       					: BOOL;  								// Zezwolenie na prace stacji sprawdzania nakrętek
    lrLidPuttedCheckHeightSV 	 					: LREAL; 								// Wysokość na której ma znajdować się stacja sprawdzania nakrętek
	lrLidPuttedCheckPosition						: LREAL;								// Pozycja sprawdzania platynki
	lrLidPuttedCheckArea							: LREAL;								// Granicy sprawdzania platynki
	bLidPuttedCheckInCameraArea1					: BOOL;									// Wózek 1 sprawdzany
	bLidPuttedCheckInCameraArea2					: BOOL;									// Wózek 2 sprawdzany
	iLidPuttedCheckProgram							: INT;	
	
	//Przygrzewaczki
	lrLidSealerPressure								: LREAL;									//	Siła zgrzewania [kg]                                              
	//Przygrzewaczka 1                              
	bLidSealerEnable								: BOOL;									// Zezwolenie na pracę podajnika 
	bLidSealerDoHoming								: BOOL; 								// Wykonanie bazowania przez przygrzewacz platynek
    bLidSealerHeaterEnable							: BOOL;								    // Zezwolenie na prace grzałki 
    iLidSealerHeatingTime							: INT	:=700;						    // Czas zgrzewania  [ms]
    iLidSealer1TempSV								: INT	:=150;							// Temperatura zadana grzałki 
	nLidSealerTempHisteresis						: INT;							    	// Histereza poprawnej temperatury grzałki (+/- *C), po jej przekroczeniu grzałka wpada w błšd
    lrLidSealerHeightPosSV							: LREAL	:=55;						    // Wysokoć na której ma znajdować się grzałka
	                                                
	//Przygrzewaczka 2                              
    bLidSealer2Enable								: BOOL;									// Zezwolenie na pracę podajnika 								// Wykonanie bazowania przez przygrzewacz platynek 
	bLidSealer2HeaterEnable							: BOOL;								    // Zezwolenie na prace grzałki 
    iLidSealer2TempSV								: INT	:=150;							// Temperatura zadana grzałki 
	
	//Przeciąganie przygrzewaczka
	bLidSealerDragingStationEnable							: BOOL;
	bLidSealerDragingStationDoHoming				: BOOL;
	bLidSealerDragingStationPrepareRun				: BOOL;
	lrLidSealerDragingStationVelocity				: LREAL	:= 100; 						// Zadana prędkosć ruchu przeciągania formatek pod zakręcarkam
	lrLidSealerDragingStationAcceleration			: LREAL	:=12;							// Przyspieszenie przeciągania
	lrLidSealerDragingStationDeceleration			: LREAL	:=15;							// Hamowanie przeciągania
	aLidSealerDragingAxisRef						: AXIS_REF;
	bLidSealerDragingHeightSet						: BOOL;	
	iLidSealerDragFormCounter						: INT;
	
	//Przeciąganie za robotem (rotacja formatek)
	bAfterRobotDragingStationEnable							: BOOL;
	bAfterRobotDragingStationDoHoming				: BOOL;
	bAfterRobotDragingStationPrepareRun				: BOOL;
	lrAfterRobotDragingStationVelocity				: LREAL	:= 100; 						// Zadana prędkosć ruchu przeciągania formatek pod zakręcarkam
	lrAfterRobotDragingStationAcceleration			: LREAL	:=12;							// Przyspieszenie przeciągania
	lrAfterRobotDragingStationDeceleration			: LREAL	:=15;							// Hamowanie przeciągania
	aAfterRobotDragingAxisRef						: AXIS_REF;
	bAfterRobotDragingHeightSet						: BOOL;	
	iAfterRobotDragFormCounter						: INT;	
	
	(*****P05_WeightCorrection******)
	lrFormWeight 									:LREAL;									// Waga formatki
	
	lrFormWeight1RFID								:LREAL;									// Waga formatki z RFID
	lrFormWeight2RFID								:LREAL;									// Waga formatki z RFID
	lrFormWeight3RFID								:LREAL;									// Waga formatki z RFID
	lrFormWeight4RFID								:LREAL;									// Waga formatki z RFID
	
	lrFormWeight5RFID								:LREAL;									// Waga formatki z RFID
	lrFormWeight6RFID								:LREAL;									// Waga formatki z RFID

	lrMass1Density									:LREAL;(*#p*)							//Gęstoć masy [g/ml]
	lrMass2Density									:LREAL;(*#p*)							//Gęstoć masy [g/ml]
	lrCupWeight										:LREAL;(*#p*)							//Waga samego kubeczka [g]
	lrWholePackageWeight							:LREAL;(*#p*)							//Waga całego opakowania bez masy (kubeczek,platynka,nakrętka) [g]
	lrWeight1MeasurmentCorrection					:LREAL;(*#p*)							//Korekta wagi zmierzonej [g]//Korekta wagi zmierzonej [g]

	iWeightCorrectionNumberOfSamples				:UINT;									// Ilość próbek dla korekty dozy

	bDispencer1WeightCorrectionEnable				:BOOL;(*#p*)							//Zezwolenie na pracę bloku korekcji, jeli przełšczy sie w tryb 
	bDispencer2WeightCorrectionEnable				:BOOL;(*#p*)							//Zezwolenie na pracę bloku korekcji, jeli przełšczy sie w tryb 
	bDispencer3WeightCorrectionEnable				:BOOL;(*#p*)							//Zezwolenie na pracę bloku korekcji, jeli przełšczy sie w tryb 
	bDispencer4WeightCorrectionEnable				:BOOL;(*#p*)							//Zezwolenie na pracę bloku korekcji, jeli przełšczy sie w tryb 
	lrWeightUpperTolerance							:LREAL;(*#p*)							//Górny zakres tolerancji wagi [g]
	lrWeightLowerTolerance							:LREAL;(*#p*)							//Zakres tolerancji wagi poniżej zadanej [g]	

	(*****P08_CapFeeder*****)
	bCapFeederDoHoming: BOOL;										// Wykonanie bazowania stacji podajnika nakrętek
	bCapFeederEnable: BOOL; 	
    lrCapFeederHeightPosSV: LREAL;									 	
	iCapFeederTimeDelayOn: INT; 										
	iCapFeederTimeDelayOff: INT; 
	iCapFeederTimeToEmptySleeveError: INT;							// Czas do alarmu pustego rękawa 

	(*****P08_CapSorter*****)
	bCapFeederGateEnable	:BOOL;									// Załączenie szlabanu podawania zamknięć 
	iCapFeederGateBlockingTime	:INT;								// Czas blokowania szlabnu podawania zamknięć
	iCapFeederCheckCountNOK	:INT;									// Zliczanie butelek bez nasadek

	//Sorter nasadek
	bCapSorterOnlyWeightOKEnable				:BOOL;
	
	//Przeciąganie formatek
	aCapSorterDragAxisRef							:AXIS_REF;								// Struktura osi napędu krokowego przeciągania	
	bCapSorterDragEnable							:BOOL;									// Zezwolenie na pracę przeciągania 
	bCapSorterDragDoHoming							:BOOL;									// Wykonanie bazowania przeciągania
	bCapSorterDragHeightSet							:BOOL;									// Wykonanie bazowania przeciągania
	lrCapSorterDragVelocity							:LREAL:=100;							// Prędkośc przeciągania
	lrCapSorterDragAcceleration						:LREAL:=12;								// Przyspieszenie przeciągania
	lrCapSorterDragDeceleration						:LREAL:=15;								// Hamowanie przeciągania
	bCapSorterDragPrepareRun						:BOOL;
	iCapSorterDragFormCounter						:INT;
	
	(*****P09_CapPuttedCheck*****)
	bCapPuttedCheckDoHoming							:BOOL;									// Wykonanie bazowania stacji sprawdzania nakrętek
	bCapPuttedCheckEnable							:BOOL; 									// Zezwolenie na prace stacji sprawdzania nakrętek
	lrCapPuttedCheckHeightPosSV						:LREAL:=69;(**) 					   	// Wysokość na której ma znajdować się stacja sprawdzania nakrętek
	bCapPuttedCheckRun								:BOOL;
	
	(****P10A_BottleDrag****) 
	bBottleDragingStationEnable						:BOOL;
	lrBottleDragingStationVelocity					:LREAL; 				
	bBottleDragingStationDoHoming					:BOOL;
	bBottleDragingStationPrepareRun					:BOOL;
	aBottleDragingAxisRef							:AXIS_REF;				
	bBottleDragingHeightSet							:BOOL;						
	
	bDelay40sAfterReset								:BOOL;
	
	(*****P10_GripperScrewer********)
	aGripperScrewer1LiftAxisRef						:AXIS_REF;//ActPos						// Struktura NC napędu podnosnika zakręcarki szczękowej
	aGripperScrewer2LiftAxisRef						:AXIS_REF;//ActPos						// Struktura NC napędu podnosnika zakręcarki szczękowej
	aGripperScrewer1AxisRef							:AXIS_REF; 								// Struktura NC napędu zakręcarki szczękowej 1
	aGripperScrewer2AxisRef							:AXIS_REF; 								// Struktura NC napędu zakręcarki szczękowej 2
	aGripperScrewer1EncoderAxisRef					:AXIS_REF; 								// Struktura NC enkodera zakręcarki szczękowej 1
	aGripperScrewer2EncoderAxisRef					:AXIS_REF; 								// Struktura NC enkodera zakręcarki szczękowej 2
	bGripperScrewerDoHoming							:BOOL;(**)								// Bazowanie stacji zakręcarki szczękowej
	bGripperScrewer1Enable							:BOOL;						// Aktywacja pierwszeh zakrecarki
	bGripperScrewer2Enable							:BOOL;						// Aktywacja drugiej zakrecarki
	bGripperScrewerFindScrew						:BOOL; 						// Aktywacja szukania gwintu	
	lrGripperScrewerFindingScrewDegree				:LREAL; 					// Kąt szukania gwintu
	iGripperScrewer1Tool							:INT;						// Wybór narzędzia (1-5), opisy w tablicy AsGripperScrewerTool	
	bGripperScrewerOption1							:BOOL;						// Otwarty chwytak przy szukaniu gwintu
	bGripperScrewerOption2							:BOOL;						// Obrót do tyłu w pozycji dociskania
	bGripperScrewerOption3							:BOOL;						// Dodatkowe zamknięcie chwytakiem przed zakręceniem 
	bGripperScrewerOption4							:BOOL;						// Szukanie gwintu w pozycji dociskania
	bGripperScrewerOption5							:BOOL;						// Szukanie gwintu z czujnikiem wysokości
	bGripperScrewerOption6							:BOOL;						// Szukanie gwintu z czujnikiem wysokości
 	bGripperScrewerOption7							:BOOL;						// Szukanie gwintu z czujnikiem wysokości
 	lrGripperScrewerVelocity						:LREAL:=6000; 				// Prędkość zakręcania
	nGripperScrewerTightTime						:INT:=100;  				// Czas przytrzymania nakrętki z zadanym momentem [ms] 
	iGripperScrewerStartDelay						:INT;						// Zwoka przed zakręcaniem			
	lrGripperScrewingTightTorque					:LREAL;  					// Nastawa momentu zakręcania [Nm]
	lrGripperScrewing2TightTorque					:LREAL;  					// Nastawa momentu zakręcania 2[Nm]
	lrGripperScrewerReadyPosition					:LREAL := 250;  			// Pozycja gotowości
	lrGripperScrewerPushingCapPosition				:LREAL := 250;  			// Pozycja docisku nakrętki 
    lrGripperScrewerScrewingCapPosition				:LREAL := 250;  			// Pozycja zakręcania nakrętki
	lrGripperScrewerFindScrewPosition				:LREAL := 250;  			// Pozycja zakręcania nakrętki
	bGripperScrewerFindScrewAdjust					: BOOL; 								// Wlaczanie dłuższego szukania  z szukaniem MIN i MAX wysokości z czujnikiem wysokości 
	lrGripperScrewerTurnoversToFullScrewed 			:LREAL;
   	lrGripperScrewerThreadPitch						:LREAL;
	lrGripperScrewerThreadTimes						:LREAL;
	
	//Chytak zakrecarki
	bGripperScrewerCatch1Homing						:BOOL;
	bGripperScrewerCatch2Homing						:BOOL;
	
	bGripperScrewerCatch1DoHoming					:BOOL;(**)								// Bazowanie stacji łapania pod zakręcarki szczękowej
	bGripperScrewer1Catch							:BOOL;  						        // Rozkaz chwytania opakowania pod zakręcarkš
	nGripperScrewerCatchHeightSV					:LREAL:=36;(*#pp*)						// Zadana wartoć pozycji bazowania stacji chwytania opakowania pod zakręcarkš

	bGripperScrewerCatch2DoHoming					:BOOL;(**)								// Bazowanie stacji łapania pod zakręcarki szczękowej
	bGripperScrewer2Catch							:BOOL;  						        // Rozkaz chwytania opakowania pod zakręcarkš	
	
	(*****P11B_CapPuttedCheck*****)
	bCapCorrectCheckDoHoming						:BOOL;									// Wykonanie bazowania stacji sprawdzania nakrętek
	bCapCorrectCheckEnable							:BOOL; 									// Zezwolenie na prace stacji sprawdzania nakrętek
	lrCapCorrectCheckHeightPosSV					:LREAL:=69;(**) 				   		// Wysokość na której ma znajdować się stacja sprawdzania nakrętek
	bCapCorrectCheckCameraEnable					:BOOL;  
	iCapCorrectCheckCameraProgram                   :INT;	
	
	(*****P13_BottleTransfer********)
	bBottleTransferEnable							:BOOL;(*#p*)         					// Właczenie robota
	nBottleTransferProgram							:UINT;(*#p*)         					// Program robota

 	bBottleTransferDoHoming							:BOOL;									// Rozkaz wykonania pozycjonowania robota
	iBottleTransferPickOffsetX						:INT;
	iBottleTransferPickOffsetY						:INT;  
	iBottleTransferPickOffsetZ						:INT;   
	iBottleTransferPick2OffsetX						:INT;
	iBottleTransferPick2OffsetY						:INT;  
	iBottleTransferPick2OffsetZ						:INT;   

	iBottleTransferPlace1OffsetX					:INT;
	iBottleTransferPlace1OffsetY					:INT;  
	iBottleTransferPlace1OffsetZ					:INT;
	iBottleTransferPlace2OffsetX					:INT;
	iBottleTransferPlace2OffsetY					:INT;
	iBottleTransferPlace2OffsetZ					:INT; 
	iBottleTransferSpeed							:INT := 2;								// predkosc robota pozioma	
	bBottleTransferInkJetEnable						:BOOL;									// Przejazd robota przez InkJet
  	bBottleTransferPickOnlyOne						:BOOL;						// Pobieranie tylko 1 opakowania
	bBottleTransferWeightEnable						:BOOL;
    iBottleTransferWeightInterval					:INT;	
	
	(***P13_BottleTransferAfterDrag***)	
	//Przeciąganie formatek 
	bBottleTransferAfterDragEnable					:BOOL;									// Zezwolenie na pracę przeciągania 
	bBottleTransferAfterDragDoHoming				:BOOL;									// Wykonanie bazowania przeciągania
	bBottleTransferAfterDragHeightSet				:BOOL;									// Wykonanie bazowania przeciągania
		
